	(*Rüstsatz 154 Rasterplattel*)
	ST03_418_B60_6: sDigInVisu;		(*  Zuführung links frei zum Ablegen ISK SP Maschine *)
	ST03_418_B60_7: sDigInVisu;		(*  Zuführung rechts frei zum Ablegen ISK SP Maschine *)

	ST03_419_B61_0: sDigInVisu;		(*  Förderband Zuführung links ISK anwesend zum Vereinzeln*)
	ST03_419_B61_1: sDigInVisu;		(*  Förderband Zuführung rechts ISK anwesend zum Vereinzeln*)
	ST03_419_B61_2: sDigInVisu;		(*  Züführung links ISK auf Übergabeposition Roboter Palettierer*)
	ST03_419_B61_3: sDigInVisu;		(*  Züführung rechts ISK auf Übergabeposition Roboter Palettierer*)

	ST03_419_Y61_5 : sValveVisu; 		(* Förderband linke Zuführung Vereinzler AST/GST *)
	ST03_419_Y61_6 : sValveVisu; 		(* Förderband rechte Zuführung Vereinzler AST/GST *)
	ST03_419_Y61_7 : sValveVisu; 		(* Förderband links/rechts Züführung Stopper AST/GST *)

	(*Rüstsatz 154pol*)

	ST03_425_B67_4: sDigInVisu;		(*  Zuführung  frei zum Ablegen ISK SP Maschine Pos.1 *)
	ST03_425_B67_5: sDigInVisu;		(*  Zuführung  frei zum Ablegen ISK SP Maschine Pos.2 *)
	ST03_425_B67_6: sDigInVisu;		(*  Zuführung  frei zum Ablegen ISK SP Maschine Pos.3 *)
	ST03_425_B67_7: sDigInVisu;		(*  ISK anwesend am Vereinzler*)

	ST03_426_B68_4: sDigInVisu;		(*  Züführung  ISK auf Übergabeposition Roboter Palettierer*)
	ST03_426_Y68_5 : sValveVisu; 		(* Förderband  Zuführung Vereinzler AST/GST *)
	ST03_426_Y68_6 : sValveVisu; 		(* Förderband  Züführung Stopper AST/GST *)


	(*Rüstsatz 160pol*)
	ST03_421_B63_4: sDigInVisu;		(*  Förderband frei zum Ablegen ISK SP Maschine Pos1 *)
	ST03_421_B63_5: sDigInVisu;		(*  Förderband frei zum Ablegen ISK SP Maschine Pos2 *)
	ST03_421_B63_6: sDigInVisu;		(*  Förderband frei zum Ablegen ISK SP Maschine Pos3 *)
	ST03_421_B63_7: sDigInVisu;		(*  ISK anwesend am Vereinzler*)
	ST03_422_B64_0: sDigInVisu;		(* Förderband Trigger Tintenstrahldrucker 1 (Lichtschranke)Rüstsatz*)
	ST03_423_B66_0: sDigInVisu;		(* Förderband Trigger Tintenstrahldrucker 2 (Lichtschranke) Rüstsatz*)
	ST03_8_B76_1: sDigInVisu;		(* Förderband Trigger Tintenstrahldrucker (Lichtschranke) 3621*)
	ST03_8_B76_2: sDigInVisu;		(* Förderband Trigger Tintenstrahldrucker (Lichtschranke) 3621*)
	ST03_422_B64_3: sDigInVisu;		(* Förderband ISK anwesend Stopper 1 Kamera*)
	ST03_423_B65_2: sDigInVisu;		(* Förderband ISK anwesend Stopper 2 Kamera*)
	ST03_423_B65_5: sDigInVisu;		(* Förderband ISK anwesend Stopper 3 Kamera*)
	ST03_422_B64_4: sDigInVisu; 		(* Zuführung ISK auf Übergabeposition Robo Palettierer*)

	ST03_422_Y64_5 : sValveVisu; 		(* Förderband  Zuführung Vereinzler AST/GST *)
	ST03_422_Y64_6 : sValveVisu; 		(* Förderband  Stopper Vereinzler AST/GST *)
	ST03_422_Y64_7 : sValveVisu; 		(* Förderband  Stopper 1 Kamera AST/GST *)
	ST03_423_Y65_6 : sValveVisu; 		(* Förderband  Stopper 2 Kamera AST/GST *)
	ST03_423_Y65_7 : sValveVisu; 		(* Förderband  Stopper 3 Kamera AST/GST *)

	ST03_33F4: sDigInVisu; 			(*Steckdosenleise Tintenstrahldrucker*)
	ST03_70U3_1: sDigInVisu; 			(*Bereit/ Im Druck Tintenstrahldrucker Frontseite*)
	ST03_70U3_2: sDigInVisu; 			(*Tank voll Tintenstrahldrucker Frontseite*)
	ST03_70U3_3: sDigInVisu; 			(*Fehler/Störung Tintenstrahldrucker Frontseite*)
	ST03_71U3_1: sDigInVisu; 			(*Bereit/ Im Druck Tintenstrahldrucker Rückseite*)
	ST03_71U3_2: sDigInVisu; 			(*Tank voll Tintenstrahldrucker Rückseite*)
	ST03_71U3_3: sDigInVisu; 			(*Fehler/Störung Tintenstrahldrucker Rückseite*)

	ST03_PLAN_70V1_1:sDigOutInVisu; 	(* Start  Bedrucken Tintenstrahldrucker Frontseite*)
	ST03_PLAN_71V1_2:sDigOutInVisu; 	(* Start  Bedrucken Tintenstrahldrucker Rückseite*)

	ST03_Y01 			: sValveVisu; 			(*1: Einschaltventil Hauptluft Tintenstrahldrucker nur bei SG-Maschine 3621*)
	ST03_S18			: sDigInVisu; 			(* ST02 Druckschalter Wartungseinheit Hauptluft min.6 bar *)
	ST03_H6 			: sDigOutInVisu; 		(* Signalsäule GR Bedruckung IO *)
	ST03_H7 			: sDigOutInVisu; 		(* Signalsäule RD Sammelstörung Bedruckung *)

	(*Rüstsatz 206pol*)

	ST03_435_B67_4: sDigInVisu;		(*  Zuführung  frei zum Ablegen ISK SP Maschine Pos.1 *)
(*	ST03_425_B67_5: sDigInVisu;		(*  Zuführung  frei zum Ablegen ISK SP Maschine Pos.2 *)
	ST03_425_B67_6: sDigInVisu;		(*  Zuführung  frei zum Ablegen ISK SP Maschine Pos.3 *) *)
	ST03_435_B67_7: sDigInVisu;		(*  ISK anwesend am Vereinzler*)

	ST03_436_B68_1: sDigInVisu;		(*  Züführung  ISK auf Übergabeposition Roboter Palettierer 1*)
	ST03_436_B68_2: sDigInVisu;		(*  Züführung  ISK auf Übergabeposition Roboter Palettierer 2*)
	ST03_437_B68_4: sDigInVisu;		(*  Züführung  ISK auf Übergabeposition Roboter Palettierer*)
	ST03_437_Y68_5 : sValveVisu; 		(* Förderband  Zuführung Vereinzler AST/GST *)
	ST03_437_Y68_6 : sValveVisu; 		(* Förderband  Züführung Stopper AST/GST *)

(*Rüstsatz92pol*)

	ST03_444_B69_4: sDigInVisu;		(*  Zuführung  frei zum Ablegen ISK SP Maschine Pos.1 *)
	ST03_444_B69_7: sDigInVisu;		(*  ISK anwesend am Vereinzler*)

	ST03_445_B70_1: sDigInVisu;		(*  Züführung  ISK auf Übergabeposition Roboter Palettierer 1*)
	ST03_445_B70_2: sDigInVisu;		(*  Züführung  ISK auf Übergabeposition Roboter Palettierer 2*)
	ST03_446_B70_4: sDigInVisu;		(*  Züführung  ISK auf Übergabeposition Roboter Palettierer*)
	ST03_446_Y70_5 : sValveVisu; 		(* Förderband  Zuführung Vereinzler AST/GST *)
	ST03_446_Y70_6 : sValveVisu; 		(* Förderband  Züführung Stopper AST/GST *)


(*Rüstsatz124pol*)

	ST03_451_B69_4: sDigInVisu;		(*  Zuführung  frei zum Ablegen ISK SP Maschine Pos.1 *)
	ST03_451_B69_7: sDigInVisu;		(*  ISK anwesend am Vereinzler*)

	ST03_452_B70_1: sDigInVisu;		(*  Züführung  ISK auf Übergabeposition Roboter Palettierer 1*)
	ST03_452_B70_2: sDigInVisu;		(*  Züführung  ISK auf Übergabeposition Roboter Palettierer 2*)
	ST03_453_B70_4: sDigInVisu;		(*  Züführung  ISK auf Übergabeposition Roboter Palettierer*)
	ST03_453_Y70_5 : sValveVisu; 		(* Förderband  Zuführung Vereinzler AST/GST *)
	ST03_453_Y70_6 : sValveVisu; 		(* Förderband  Züführung Stopper AST/GST *)

(*Rüstsatz46pol*)

	ST03_461_B69_4: sDigInVisu;		(*  Zuführung  frei zum Ablegen ISK SP Maschine Pos.1 *)
	ST03_461_B69_7: sDigInVisu;		(*  ISK anwesend am Stopper*)

	ST03_462_B70_0: sDigInVisu;		(*   Förderband  ISK anwesend Wender*)
	ST03_462_B70_1: sDigInVisu;		(*  Züführung  ISK auf Übergabeposition Roboter Palettierer Lageerkennung 1*)
	ST03_462_B70_2: sDigInVisu;		(*  Züführung  ISK auf Übergabeposition Roboter Palettierer Lageerkennung 2*)
	ST03_463_B70_7: sDigInVisu;		(*  Züführung  ISK auf Übergabeposition Roboter Palettierer *)

	ST03_464_Y71_0 : sValveVisu; 		(* Förderband  Zuführung Vereinzelner Wendestation AST/GST *)
	ST03_464_Y71_1 : sValveVisu; 		(* Förderband  Zuführung Zylinder Vakuumdüsen AST/GST *)
	ST03_464_Y71_2 : sValveVisu; 		(* Förderband  Zuführung Wendestation Einlauf / Auslauf *)
	ST03_464_Y71_3 : sValveVisu; 		(* Förderband  Zuführung Vereinzler AST/GST *)
	ST03_464_Y71_4 : sValveVisu; 		(* Förderband  Zuführung Stopper AST/GST *)
	ST03_464_Y71_5 : sValveVisu; 		(* Förderband  Zuführung Vakuumdüsen EIN/AUS *)
	ST03_464_B71_6: sDigInVisu;		(* Förderband  Vakuum vorhanden *)
 	ST03_464_B71_7: sDigInVisu;		(*Förderband  Staustrecke mitte voll *)

(*Rüstsatz NOX 5+6 pol*)

	ST03_4x2_B69_0: sDigInVisu;		(*Zuführung frei zum Ablegen ISK SP Maschine *)
	ST03_4x2_B69_5: sDigInVisu;		(* ISK anwesend am Stopper *)

	ST03_4x3_B70_0: sDigInVisu;		(* ISK anwesend Übergabeposition Stopper*)
	ST03_4x3_B70_1: sDigInVisu;		(* ISK anwesend Übergabeposition*)

	ST03_4x3_Y70_5 : sValveVisu; 	(* Zuführung Vereinzler AST/GST *)
	ST03_4x3_Y70_6 : sValveVisu; 	(* Zuführung Stopper AST/GST *)
	ST03_4x3_Y70_7 : sValveVisu; 	(* Zuführung Stopper Übergabeposition AST/GST *)

(*Rüstsatz NOX 4 pol*)
	ST03_491_B69_0: sDigInVisu;		(*  Zuführung  frei zum Ablegen ISK SP Maschine*)
	ST03_491_B69_5: sDigInVisu;		(*  ISK anwesend am Stoper*)
	ST03_491_B69_7: sDigInVisu;		(*  ISK auf Abholposition Robi*)

	ST03_492_Y70_0 : sValveVisu; 		(* Förderband  Zuführung Vereinzler AST/GST *)
	ST03_492_Y70_1 : sValveVisu; 		(* Förderband  Züführung Stopper AST/GST *)

(*Rüstsatz 88 pol*)
	ST03_501_B69_0: sDigInVisu;		(*  Zuführung  frei zum Ablegen ISK SP Maschine*)

	ST03_501_B69_5: sDigInVisu;		(*  ISK anwesend am Vereinzler*)
	ST03_501_B69_6: sDigInVisu;		(*  ISK anwesend am Stoper*)
	ST03_501_B69_7: sDigInVisu;		(*  ISK auf Abholposition Robi*)

	ST03_502_B70_0: sDigInVisu;		(*  ISK Lageerkennung*)
	ST03_502_Y70_1 : sValveVisu; 		(* Förderband  Zuführung Vereinzler AST/GST *)
	ST03_502_Y70_2 : sValveVisu; 		(* Förderband  Züführung Stopper AST/GST *)

(*Rüstsatz 7 pol*)
	ST03_512_XG1:    sDigInVisu;			(*  ISK in Rinne*)
	ST03_514_B71_7: sDigInVisu;		(*  Führungsschiene frei zum schwenken*)

	ST03_513_B70_4: sDigInVisu;		(*  ISK anwesend am Stoper*)
	ST03_513_B70_7: sDigInVisu;		(*  ISK auf Übergabeposition 1*)

	ST03_514_B71_2: sDigInVisu;		(*  ISK auf Übergabeposition 2*)
	ST03_514_B71_5: sDigInVisu;		(*  ISK auf Übergabeposition 3*)
	ST03_514_B71_6: sDigInVisu;		(*  ISK auf Übergabeposition 4*)

	ST03_515_Y72_0 : sValveVisu; 		(* SK Klemmen in Rinne AST/GST *)
	ST03_515_Y72_1 : sValveVisu; 		(* Rinne schwenkern AST/GST *)
	ST03_515_Y72_2 : sValveVisu; 		(* Führungsschiene  Zuführung Vereinzler AST/GST *)
	ST03_515_Y72_3 : sValveVisu; 		(* Führungsschiene  Zuführung Stopper AST/GST *)
	ST03_515_Y72_4 : sValveVisu; 		(* Übergabeposition Stopper 1  AST/GST *)
	ST03_515_Y72_5 : sValveVisu; 		(* Übergabeposition Stopper 2  AST/GST *)
	ST03_515_Y72_6 : sValveVisu; 		(* Übergabeposition Stopper 3  AST/GST *)

(*Rüstsatz 88 pol AMG*)
	ST03_521_B69_0: sDigInVisu;			(*Zuführung  frei zum Ablegen ISK SP Maschine*)

	ST03_521_B69_6: sDigInVisu;			(*ISK anwesend am Stopper*)
	ST03_521_B69_7: sDigInVisu;			(*ISK Lageerkennung links*)

	ST03_522_B70_0: sDigInVisu;			(*ISK Lageerkennung rechts*)
	ST03_522_Y70_1 : sValveVisu; 		(*Zuführung Vereinzler AST/GST *)
	ST03_522_Y70_2 : sValveVisu; 		(*Züführung Stopper AST/GST*)

(*Rüstsatz 120 pol *)
	ST03_531_B69_0: sDigInVisu;			(*Zuführung  frei zum Ablegen ISK SP Maschine*)

	ST03_531_B69_6: sDigInVisu;			(*ISK anwesend am Stopper*)
	ST03_531_B69_7: sDigInVisu;			(*ISK rechts Lageerkennung*)

	ST03_532_B70_0: sDigInVisu;			(*ISK links Lageerkennung *)
	ST03_532_Y70_1 : sValveVisu; 		(*Zuführung Vereinzler AST/GST *)
	ST03_532_Y70_2 : sValveVisu; 		(*Züführung Stopper AST/GST*)

(*Rüstsatz 21 pol *)
	ST03_536_B69_0: sDigInVisu;			(*Zuführung  frei zum Ablegen ISK SP Maschine*)

	ST03_536_B69_6: sDigInVisu;			(*ISK anwesend am Stopper*)
	ST03_536_B69_7: sDigInVisu;			(*ISK anwesend an Abholposition*)

	ST03_537_B70_0: sDigInVisu;			(*ISK Lageerkennung *)
	ST03_537_Y70_1 : sValveVisu; 		(*Zuführung Vereinzler AST/GST *)
	ST03_537_Y70_2 : sValveVisu; 		(*Züführung Stopper AST/GST*)

(*Rüstsatz 191 pol *)
	ST03_541_B69_0: sDigInVisu;			(*Zuführung  frei zum Ablegen ISK SP Maschine*)

	ST03_541_B69_6: sDigInVisu;			(*ISK anwesend am Stopper*)
	ST03_541_B69_7: sDigInVisu;			(*ISK rechts Lageerkennung*)

	ST03_542_B70_0: sDigInVisu;			(*ISK links Lageerkennung*)
	ST03_542_Y70_1 : sValveVisu; 		(*Zuführung Vereinzler AST/GST *)
	ST03_542_Y70_2 : sValveVisu; 		(*Züführung Stopper AST/GST*)

(*Rüstsatz  72pol *)
	ST03_546_B69_0: sDigInVisu;			(*Zuführung  frei zum Ablegen ISK SP Maschine*)

	ST03_546_B69_6: sDigInVisu;			(*ISK anwesend am Stopper*)
	ST03_546_B69_7: sDigInVisu;			(*ISK rechts Lageerkennung*)

	ST03_547_B70_0: sDigInVisu;			(*ISK links Lageerkennung*)
	ST03_547_Y70_1 : sValveVisu; 		(*Zuführung Vereinzler AST/GST *)
	ST03_547_Y70_2 : sValveVisu; 		(*Züführung Stopper AST/GST*)

(*Rüstsatz 48 pol *)
	ST03_551_B69_0: sDigInVisu;			(*Zuführung  frei zum Ablegen ISK SP Maschine*)

	ST03_551_B69_6: sDigInVisu;			(*ISK anwesend am Stopper*)
	ST03_551_B69_7: sDigInVisu;			(*ISK rechts Lageerkennung*)

	ST03_552_B70_0: sDigInVisu;		(*ISK links Lageerkennung*)
	ST03_552_Y70_1 : sValveVisu; 		(*Zuführung Vereinzler AST/GST *)
	ST03_552_Y70_2 : sValveVisu; 		(*Züführung Stopper AST/GST*)

(*Rüstsatz 268 pol *)
	ST03_556_B69_0: sDigInVisu;		(*Zuführung  frei zum Ablegen ISK SP Maschine*)

	ST03_556_B69_5: sDigInVisu;		(* Führungsschiene Überwachung Staustrecke*)
	ST03_556_B69_6: sDigInVisu;		(*ISK anwesend am Stopper*)
	ST03_556_B69_7: sDigInVisu;		(*ISK anwesend an Abholposition*)

	ST03_557_Y70_1 : sValveVisu; 		(*Zuführung Vereinzler AST/GST *)
	ST03_557_Y70_2 : sValveVisu; 		(*Züführung Stopper AST/GST*)

(*Rüstsatz 268 pol Rasterplatte======================================================================================*)
	ST03_562_B69_0: sDigInVisu;		(*Zuführung 1 frei zum schwenken*)
	ST03_562_B69_6: sDigInVisu;		(*Zuführung 1 ISK anwesend am Stopper*)
	ST03_562_B67_7: sDigInVisu;		(*Zuführung 1 ISK auf Übergabepos. Robi*)

	ST03_563_B70_0: sDigInVisu;		(*Zuführung 2 frei zum schwenken*)
	ST03_563_B70_6: sDigInVisu;		(*Zuführung 2 ISK anwesend am Stopper*)
	ST03_563_B70_7: sDigInVisu;		(*Zuführung 2 ISK auf Übergabepos. Robi*)

	ST03_564_Y71_0: sValveVisu; 		(*Zuführung 1 Vereinzler AST/GST *)
	ST03_564_Y71_1: sValveVisu; 		(*Zuführung 1 Stopper AST/GST *)
	ST03_564_Y71_2: sValveVisu; 		(*Zuführung 2 Vereinzler AST/GST *)
	ST03_564_Y71_3: sValveVisu; 		(*Zuführung 2 Stopper AST/GST *)
	ST03_564_Y71_4: sValveVisu; 		(* ISK Klemmer AST/GST *)
	ST03_564_Y71_5: sValveVisu; 		(* Rinne schwenkern AST/GST *)

	ST03_565_B72_0: sDigInVisu;		(* ISK 1 in Klemmer*)
	ST03_565_B72_1: sDigInVisu;		(* ISK 2 in Klemmer*)

(*Rüstsatz 33 pol Rasterplatte======================================================================================*)
	ST03_571_B69_0	: sDigInVisu;		(* Zuführung  Pos 1 frei zum Ablegen ISK SP Maschine*)
	ST03_571_B69_1	: sDigInVisu;		(* Zuführung  Pos 2 frei zum Ablegen ISK SP Maschine*)

	ST03_571_B69_6	: sDigInVisu;		(* ISK anwesend am Stopper*)
	ST03_571_B69_7	: sDigInVisu;		(* ISK anwesend an Abholposition*)

	ST03_572_Y70_0	: sValveVisu; 		(* Zuführung Vereinzler AST/GST *)
	ST03_572_Y70_1	: sValveVisu; 		(* Züführung Stopper AST/GST *)

(*---------------------------------------------------------------------------
  Station08
  ---------------------------------------------------------------------------*)


	ST08_170_Q2 : sDigInVisu; (* Bandstrecken Station 8 Motorschutz i.O. *)
	ST08_170_M : sDigInVisu; (* Bandstrecken Station 8 Thermokontakt i.O. *)

	ST08_400_B50_0 : sDigInVisu; (* Traystapel vor Vereinzeler Einlaufband hinten *)
	ST08_401_B50_5 : sDigInVisu; (* Traystapel vor Vereinzeler Einlaufband mitte *)
	ST08_402_B51_2 : sDigInVisu; (* Traystapel vor Vereinzeler Einlaufband vorne *)
	ST08_402_B51_4 : sDigInVisu; (* Luftzone 1 *)
	ST08_402_B51_5 : sDigInVisu; (* Luftzone 2 *)
	ST08_404_B52_2 : sDigInVisu; (* Traystapel in Ablageposition Isokörper *)
	ST08_404_B52_3 : sDigInVisu; (* Traystapel richtig eingelegt Isokörper *)
	ST08_406_B54_0 : sDigInVisu; (* Tray in Zwischenp. Entnahme Isokörper (Bandende) *)
	ST08_406_B54_3 : sDigInVisu; (* Tray in Ausheber. Entnahme Isokörper (Bandende) *)
	ST08_406_B54_6 : sDigInVisu; (* Tray aus Entnahme ausgelaufen (Bandende) *)
	ST08_407_B55_1 : sDigInVisu; (* Tray aus entnahme ausgelaufen STN8 *)
	ST08_407_B55_4 : sDigInVisu; (* Tray in Aufstapelposition eingelaufen STN8 *)
	ST08_409_B55_5 : sDigInVisu; (* Auslaufrollenbahn voll STN8 *)

	ST08_412_B58_4: sDigInVisu;		(*  Rüstsatz Förderband frei zum Ablegen ISK von SP Maschine Position 1 *)
	ST08_412_B58_5: sDigInVisu;		(*  Rüstsatz Förderband frei zum Ablegen ISK von SP Maschine Position 2 *)
	ST08_412_B58_6: sDigInVisu;		(*  Rüstsatz Förderband frei zum Ablegen ISK von SP Maschine Position 3 *)
	ST08_412_B58_5_35pol: sDigInVisu;		(*  Lageerkennung links *)
	ST08_412_B58_6_35pol: sDigInVisu;		(*  Lageerkennung rechts *)
	ST08_412_B58_7: sDigInVisu;		(*  Rüstsatz Förderband ISK anwesend zum Vereinzeln *)
	ST08_412_B59_0: sDigInVisu;		(*  Rüstsatz Förderband ISK auf Übergabeposition Roboter Verpackung *)

	ST08_169_K1 : sDigOutInVisu; (* Bandantrieb 1 Einlauf Trays Ein *)
	ST08_169_K2 : sDigOutInVisu; (* Bandantrieb 4 Auslauf leere Trays Ein *)
	ST08_170_K1 : sDigOutInVisu; (* Bandantrieb 2 Hubquereinheit Trays Ein *)
	ST08_170_K2 : sDigOutInVisu; (* Bandantrieb 3 Hubquereinheit Trays Ein *)

	ST08_400_Y50_0 : sValveVisu; (* Stopper Traystapel Einlaufb. hinten links + rechts AST *)
	ST08_400_Y50_2 : sValveVisu; (* Stopper Traystapel Einlaufb. mitte links + rechts AST *)
	ST08_402_Y50_4 : sValveVisu; (* Stopper Traystapel Einlaufb. vorne links + rechts AST *)
	ST08_403_Y50_6 : sValveVisu; (* Vakuum 1 Einlauf STN8 AST *)
	ST08_403_Y50_7 : sValveVisu; (* Vakuum 2 Einlauf STN8 AST *)
	ST08_405_Y51_0 : sValveVisu; (* Hubtüre 2 Einlauf Isokörper STN8 AST *)
	ST08_404_Y51_6 : sValveVisu; (* Stopper Traystapel Isokörper AST *)
	ST08_406_Y51_2 : sValveVisu; (* Hubtüre 3 STN8 AST *)
	ST08_407_Y51_4 : sValveVisu; (* Hubtüre 4 Auslauf STN8 AST *)
	ST08_404_Y52_0 : sValveVisu; (* Hub Bandstrecke AST *)
	ST08_406_Y52_3 : sValveVisu; (* Ausheber Trays Entnahmepos. Isok. STN8 GST *)
	ST08_401_Y52_4 : sValveVisu; (* Traystapel schieben hinte AST *)
	ST08_400_Y52_5 : sValveVisu; (* Stopper links + rechts Traystapel Auslaufband einfahren *)
	ST08_402_Y52_6 : sValveVisu; (* Traystapel schieben mitte AST *)
	ST08_402_Y52_7 : sValveVisu; (* Traystapel schieben vorne AST *)
	ST08_404_Y53_0 : sValveVisu; (* Abstapelzylinder 1 Isokörper AST *)
	ST08_404_Y53_2 : sValveVisu; (* Abstapelzylinder 2 Isokörper AST *)
	ST08_405_Y53_4 : sValveVisu; (* Rückhaltezylinder li+re Traystapel Isokörper AST *)
	ST08_408_Y54_0 : sValveVisu; (* Rückhaltezylinder li.+re. Auslauf STN8 AST *)
	ST08_408_Y54_2 : sValveVisu; (* Abstapelzylinder 1 STN8 AST *)
	ST08_408_Y54_4 : sValveVisu; (* Abstapelzylinder 2 STN8 AST *)

	ST08_412_Y55_0 : sValveVisu; (* Rüstsatz Förderband Vereinzelner *)
	ST08_412_Y55_2 : sValveVisu; (* Rüstsatz Förderband Stopper *)

	ST08_180_M1 		: sDigInVisu; (* Abstapeln *)
	ST08_185_M1 		: sDigInVisu; (* Aufstapeln *)
	ST08_190_M1 		: sDigInVisu; (* Tray ausheben *)

END_STRUCT
END_TYPE

(* Data type in System/LoginDialog *)
TYPE sVisuLoginDialog :
STRUCT

	LoginKeyPad			: sNumericKeypad;
	btn_Login			: sButtonVisu;
	btn_LogOut			: sButtonVisu;
	btn_ChangeUserData	: sButtonVisu;
	btn_ChangePassword	: sButtonVisu;

	ShowEditFields		: BOOL;
	UserListIndex		: INT;

	UserEdit			: sUserData;

END_STRUCT
END_TYPE

(* POU pBasic/PLC_PRG, ST *)
PROGRAM PLC_PRG
VAR_OUTPUT
	GlobalHomePos		: BOOL;
END_VAR
VAR
	DW_alive			: DINT:=0;
	TimeStart			: TIME;
	TimeEnd				: TIME;
	fb_ton_startHYDRA	: TON;
END_VAR
DW_alive:=DW_alive+1;
TimeStart:=TIME();

BusDiagnosis();
(*LngHandler();*)
IOSimulation();
ErrorHandler.ClearAll(sVisu:=Visu.ErrorHandler);
MessageHandler.ClearAll(sVisu:=Visu.Message);
IF	ProcessMessage01 = '' OR ProcessMessage02 = '' OR
	ModeSelect.Mode<=MODE_MANUAL THEN
	ProcessMessage01:='EMPTY';
	ProcessMessage02:='EMPTY';
END_IF

ModeSelect(	sVisu				:=Visu.ModeSelect,
			ControlOn			:= ST00_200_A1_A1.BitInToCheck,
 			SafetyDoorOk		:= gReadyForControlOn,
			MainValveOk			:= ST00_350_B20_0.BitInToCheck OR		SpecialMode03.State=STATE_RUN(* @@@ *),
			EmergencyOk			:= ST00_200_A1_A1.BitInToCheck,
			BusControlState		:= STATE_OK,
			UserOK				:= TRUE,
			AutoCycleEnd 		:= CheckSFCInInit.AllSeqInInit,
			SpecialCycleEnd 	:= CallSpecialModeSFCs.AllSpecialModeSFCInInit,
			HomePosRunEnd 		:= PLC_PRG.GlobalHomePos AND HomePositionSFC.State=STATE_WAIT,
			AllDoorsClosed 		:= TRUE,
			EnableFromPrevMach	:= TRUE,
			EnableFromNextMach	:= TRUE,
			ProtecKeyNotIn		:= TRUE,
			ProtecNotBridged	:= TRUE,
			Enable 			    := TRUE,
			Reset 				:= FALSE,
					);

gResetAll:=ModeSelect.QReset;

CallGeneralFunctions();
(* Spezialfunktion: *)
(* Disconnect Scanner TCPIP-Gateway *)
gBasicManualMode:=ModeSelect.BasicManualMode;

(*----------------------------------------------------------------------------
 Main-Program
 ----------------------------------------------------------------------------*)

ST_UPS(b_Ups := TRUE);
ST_CPU();
ST_AutoCheckIn( i_IntervalDay:=7 );
ST_MainMenue();
ST_Path();
ST_MinExit();
ST_ReadXmlLine();
ST_ReadXmlLineMsg();
ST_SaveAndLoad();
ST_Lng();

fb_ton_startHYDRA(IN:=TD.ArtNo <> '',PT:=t#5s);
IF fb_ton_startHYDRA.Q THEN						(*Textdateien erst nach Einlesen der Typdaten (Maschinennummer>0) + 5 sekündiger Verzögerung schreiben/lesen*)

	(***Für HYDRA 8****************************************)
	ST_Hydra8();

	FbExportHydraString(s_Path:= 'C:\MPDV\AIP2\spool\',
					st_data:=st_Hydra8Data,
					s_system_time:=gVarStrSystemTime,
					sDateiName:= 'Eingang.txt',
					bKopiereDateiAufServer:=FALSE,
					sToolPath := s_tools_path,
					tStartTime:= T#5S);

	ST_ImportHydraString(s_Path:= 'C:\MPDV\AIP2\spool\',
						sDateiName:= 'Ausgang.txt',
						tStartTime := T#5S);

END_IF

IF gInitOk AND ST_Path.Done THEN

	ImpExp_UD(path:= s_ud_path,filename:='UserData.xml');

	UserLoginHandler(sVisu:= Visu.LoginHandler,UserList:=UD.UserList);
	TDHandler(TDActivationAlowed:= ModeSelect.Mode<=MODE_MANUAL ,sVisu:=sTDHandler);
	MPHandler(sVisu:=sMPHandler);
	MP_ShiftHandler();

	ListHomeNOK(Clear:=TRUE);
	gHomeOk:=TRUE;
	_CallFBs();

	GlobalHomePos:=gHomeOk (*AND gHomePosSFCDone*);


	_CallSFCs();
	_CallPRGs();
	CheckSFCInInit();

ELSE
	gInitCollect:=TRUE;
	_CallInit();
	gInitOk:=gInitCollect;
 (* Spezialfunktion: *)
END_IF (*gInitOk=TRUE*)

(*------------- Main-Program-End -------------------------------------------*)

ErrorHandler.HandleErrors(sVisu:=Visu.ErrorHandler);
ErrorHandler.VisuUpdate(sVisu:=Visu.ErrorHandler);
MessageHandler.VisuUpdate(sVisu:=Visu.Message);

TimeEnd:=TIME();

(*END Program -----------------------------------------------------------------*)
END_PROGRAM

(* POU System/BusDiagnosis/BusDiagnosis, ST *)
PROGRAM BusDiagnosis
VAR

	EtheCatMasterAmsNetId 		AT %I* 	: ARRAY[0..5] OF USINT;	(* AmsNetId of EtherCat Mater *)


	GetConfSlaves				: FB_EcGetConfSlaves;			(* Read all Configured Informations of Master *)
	GetScannedSlaves			: FB_EcGetScannedSlaves;
	GetAllSlaveStates			: FB_EcGetAllSlaveStates;

	ConfSlaveInfo 				: ARRAY[1..NoOfMaxSlaves] OF ST_EcSlaveConfigData;
	ScannedSlaveInfo 			: ARRAY[1..NoOfMaxSlaves] OF ST_EcSlaveScannedData;
	ScannedSlaveInfoTemp 		: ARRAY[1..NoOfMaxSlaves] OF ST_EcSlaveScannedData;

	SlaveStates					: ARRAY[1..NoOfMaxSlaves] OF ST_EcSlaveState;
	SlaveStatesTemp			: ARRAY[1..NoOfMaxSlaves] OF ST_EcSlaveState;
	StringSlaveStates			: ARRAY[1..NoOfMaxSlaves] OF STRING(80);


	FirstStart					: BOOL;

	WorkIdx					: DINT;
	ForIdx						: DINT;

END_VAR
VAR CONSTANT
	NoOfMaxSlaves				: DINT := 100;
END_VAR
(* Get EtherCat Config - ONCE after RESET *)
IF 	NOT FirstStart THEN
	GetConfSlaves.bExecute:=TRUE;
	FirstStart:=TRUE;
END_IF

(* Get actual EtherCat - Scan *)
CASE WorkIdx OF
0: (* Init *)
	WorkIdx:=1;
1: (* Start Getting Bus Scan *)
	GetScannedSlaves.bExecute:=TRUE;
	IF 	GetScannedSlaves.bBusy THEN
		WorkIdx:=2;
	END_IF
2:
	IF 	NOT GetScannedSlaves.bBusy THEN
		WorkIdx:=3;
		ScannedSlaveInfo:=ScannedSlaveInfoTemp;
	END_IF

3:(* Get Salve States *)
	GetAllSlaveStates.bExecute:=TRUE;
	IF 	GetAllSlaveStates.bBusy THEN
		WorkIdx:=4;
	END_IF
4:
	IF 	NOT GetAllSlaveStates.bBusy THEN
		WorkIdx:=5;
		SlaveStates:=SlaveStatesTemp;
		FOR ForIdx:=1 TO NoOfMaxSlaves DO
			StringSlaveStates[ForIdx]:=F_ConvSlaveStateToString(SlaveStates[ForIdx]);
		END_FOR
	END_IF
5: (* End of operation *)
	WorkIdx:=0;
END_CASE

GetConfSlaves(
	sNetId					:= GetAmsNetIdString(EtheCatMasterAmsNetId),
	pArrEcConfSlaveInfo		:= ADR(ConfSlaveInfo),
	cbBufLen				:= SIZEOF(ConfSlaveInfo),
);

GetConfSlaves.bExecute:=FALSE;

GetScannedSlaves(
	sNetId						:= GetAmsNetIdString(EtheCatMasterAmsNetId),
	pArrEcScannedSlaveInfo	:= ADR(ScannedSlaveInfoTemp),
	cbBufLen					:= SIZEOF(ScannedSlaveInfoTemp),
 );

GetScannedSlaves.bExecute:=FALSE;

GetAllSlaveStates(
	sNetId						:= GetAmsNetIdString(EtheCatMasterAmsNetId),
	pStateBuf					:= ADR(SlaveStatesTemp),
	cbBufLen					:= ADR(SlaveStatesTemp),
 );

GetAllSlaveStates.bExecute:=FALSE;
END_PROGRAM

(* POU System/BusDiagnosis/GetAmsNetIdString, ST *)
FUNCTION GetAmsNetIdString : STRING
VAR_INPUT
		EtheCatMasterAmsNetId : ARRAY[0..5] OF USINT;
END_VAR
VAR
	Idx : DINT;
END_VAR
GetAmsNetIdString:='';

FOR Idx:=0 TO 5 DO
	GetAmsNetIdString:=CONCAT(GetAmsNetIdString, USINT_TO_STRING(EtheCatMasterAmsNetId[Idx]));
	IF 	Idx<>5 THEN
		GetAmsNetIdString:=CONCAT(GetAmsNetIdString,'.');
	END_IF
END_FOR
END_FUNCTION

(* POU Stations/ST_00/ST00_PRGs/IOSimulation, ST *)
PROGRAM IOSimulation
VAR

END_VAR
SystemTaskInfoArr[1].cycleTimeExceeded;
SystemTaskInfoArr[1].lastExecTime;
END_PROGRAM

(* POU System/Error_and_Message/ErrorHandler, ST *)
PROGRAM ErrorHandler
VAR
	TempErrorArray					: sErrorHandlerVisu;
	TempErrorArrayLastCycle 		: sErrorHandlerVisu;
	TempErrorArrayLastCycleQuitt 	: sErrorHandlerVisu;
	Idx								: DINT;

	TempError						: BOOL;
	TempWarning					: BOOL;
	TempInfo						: BOOL;
	POS							: INT;
	i								: INT;

	(* Variable for ErrorHistory Handling *)
	Idx_Akt							: DINT;
	Idx_Last						: DINT;
	ErrorPresent						:BOOL;

	CompareValue					:DINT;

	(* Variables for ErrorLog.CSV *)
	ErrorLogBuffer				: ARRAY[0..100] OF ErrorStruct;
	EmptyError					: ErrorStruct;
	ErrorToLog					: ErrorStruct;
	ErrorToQuitt					: ErrorStruct;

	StepExportError				: DINT;

	(* CSV Config *)
	ColIdx						: DINT;
	DataType					: DataTypeDef;
	CSVConfig  					: ARRAY[1..20] OF CSV_Config;
	CSVConfigDone				: BOOL :=FALSE;
	ErrorExport					: CSVExport_AppendLineWithVarConfig;				(*Daten in CSV-Datei exportieren*)
END_VAR
VAR_INPUT
	ErrorLogFileName			: STRING(255) := ''; (* Filename with Path e.g. 'C:\ErrorLog.csv' *)
	ErrorToAdd					: ErrorStruct;
END_VAR
VAR_OUTPUT
	bOutError					: BOOL;
	bOutWarning				: BOOL;
	bOutInfo					: BOOL;
END_VAR
VAR_IN_OUT
	sVisu						: sErrorHandlerVisu;
END_VAR
;
END_PROGRAM
ACTION AddError:
FOR Idx:=0 TO NO_OF_ERRORS
DO

	IF TempErrorArray.Error[Idx].No=0
	THEN

		FOR i:=0 TO 5 DO	(*Leerstellen entfernen*)
			POS:=0;
			POS := FIND (ErrorToAdd.Text,'$R');
			IF POS <> 0 THEN
				ErrorToAdd.Text := DELETE (ErrorToAdd.Text,1,POS);
			END_IF
			POS:=0;
			POS := FIND (ErrorToAdd.Text,'$N');
			IF POS <> 0 THEN
				ErrorToAdd.Text := DELETE (ErrorToAdd.Text,1,POS);
			END_IF
		END_FOR

		TempErrorArray.Error[Idx]:=ErrorToAdd;
			CASE TempErrorArray.Error[Idx].Typ OF
				0: TempErrorArray.Error[Idx].LineColor:=color.salmon;
				1: TempErrorArray.Error[Idx].LineColor:=color.orange;
				2: TempErrorArray.Error[Idx].LineColor:=color.lightblue;
			END_CASE
		EXIT;
	END_IF
END_FOR
END_ACTION
ACTION ClearAll:
FOR Idx:=0 TO NO_OF_ERRORS
DO
	TempErrorArray.Error[Idx].No:=0;
	TempErrorArray.Error[Idx].No:=0;
	TempErrorArray.Error[Idx].DateTime:=DINT_TO_DT(0);
	TempErrorArray.Error[Idx].Text:='';
	TempErrorArray.Error[Idx].Typ:=0;
	TempErrorArray.Error[Idx].Station:=0;
	TempErrorArray.Error[Idx].Prio:=0;
	TempErrorArray.Error[Idx].QuitAddr:=0;
END_FOR
END_ACTION
ACTION HandleErrors:
TempError			:= FALSE;
TempWarning		:= FALSE;
TempInfo			:= FALSE;

FOR Idx:=0 TO NO_OF_ERRORS
DO
	IF TempErrorArray.Error[Idx].No<>0 AND TempErrorArray.Error[Idx].Typ=0 AND NOT TempError
	THEN
		TempError:=TRUE;
	END_IF
	IF TempErrorArray.Error[Idx].No<>0 AND TempErrorArray.Error[Idx].Typ=1 AND NOT TempWarning
	THEN
		TempWarning:=TRUE;
	END_IF
	IF TempErrorArray.Error[Idx].No<>0 AND TempErrorArray.Error[Idx].Typ=2 AND NOT TempInfo
	THEN
		TempInfo:=TRUE;
	END_IF
END_FOR

bOutError:=TempError;
bOutWarning:=TempWarning;
bOutInfo:=TempInfo;

(*Eintrag in die Errorlog, wenn der Fehler wieder weggeht-----------------------------------------------------------------------------------------------------------------*)
IF MEMCMP(ADR(TempErrorArray.Error), ADR(TempErrorArrayLastCycleQuitt.Error), SIZEOF(TempErrorArray.Error))<>0 THEN
	ErrorToQuitt:=EmptyError;
	FOR Idx_Akt:=0 TO NO_OF_ERRORS DO

		FOR Idx_Last:=0 TO NO_OF_ERRORS DO
			IF	(*TempErrorArrayLastCycleQuitt.Error[Idx_Akt].DateTime = TempErrorArray.Error[Idx_Last].DateTime AND*)
				TempErrorArrayLastCycleQuitt.Error[Idx_Akt].Text = TempErrorArray.Error[Idx_Last].Text OR
				(*Ausnahmen*)
				FIND(TempErrorArrayLastCycleQuitt.Error[Idx_Akt].Text, 'MessageHandler') >0 OR
				FIND(TempErrorArrayLastCycleQuitt.Error[Idx_Akt].Text, 'TD') >0 OR
				FIND(TempErrorArrayLastCycleQuitt.Error[Idx_Akt].Text, 'Mode') >0 OR
				FIND(TempErrorArrayLastCycleQuitt.Error[Idx_Akt].Text, 'LoginHandler') >0 THEN
				EXIT;
			END_IF
		END_FOR

		IF 	Idx_Last >NO_OF_ERRORS THEN
			ErrorToQuitt:=TempErrorArrayLastCycleQuitt.Error[Idx_Akt];
			ErrorToQuitt.DateTime:=gVarDTSystemtime;
			ErrorToQuitt.Text:=CONCAT('quitt ',ErrorToQuitt.Text);

			IF ErrorLogFileName<>'' THEN
				FOR Idx:= 100 TO 2 BY -1 DO
					ErrorLogBuffer[Idx]:=ErrorLogBuffer[Idx-1];
				END_FOR
				ErrorLogBuffer[1]:=ErrorToQuitt;
			END_IF
		END_IF

	END_FOR
END_IF
TempErrorArrayLastCycleQuitt:= TempErrorArray;
(*-------------------------------------------------------------------------------------------------------------------------------------------------------------------------------------------------------*)

(* Handle Error History *)

IF MEMCMP(ADR(TempErrorArray.Error), ADR(TempErrorArrayLastCycle.Error), SIZEOF(TempErrorArray.Error))<>0
THEN
	FOR Idx_Akt:=0 TO NO_OF_ERRORS
	DO
		ErrorPresent:=FALSE;
		FOR Idx_Last:=0 TO NO_OF_ERRORS
		DO
			CompareValue:=MEMCMP(ADR(TempErrorArray.Error[Idx_Akt].DateTime), ADR(TempErrorArrayLastCycle.Error[Idx_Last].DateTime), SIZEOF(TempErrorArray.Error[Idx_Akt].DateTime));
			IF TempErrorArray.Error[Idx_Akt].DateTime = TempErrorArrayLastCycle.Error[Idx_Last].DateTime
			THEN
				ErrorPresent:=TRUE;
				EXIT;
			END_IF
		END_FOR
		(* Error is not present in List *)
		IF NOT ErrorPresent AND TempErrorArray.Error[Idx_Akt].No<>0
		THEN
			(* Add To ErrorHistory *)
			FOR Idx:= 500 TO 2 BY -1
			DO
				ErrorHistory[Idx]:=ErrorHistory[Idx-1];
			END_FOR
			ErrorHistory[1]:=TempErrorArray.Error[Idx_Akt];
			(* Add To Error Log Buffer *)
			IF ErrorLogFileName<>''
				THEN
				FOR Idx:= 100 TO 2 BY -1
				DO
					ErrorLogBuffer[Idx]:=ErrorLogBuffer[Idx-1];
				END_FOR
				ErrorLogBuffer[1]:=TempErrorArray.Error[Idx_Akt];
			END_IF

		END_IF
	END_FOR
END_IF

TempErrorArrayLastCycle:= TempErrorArray;


IF visu.ErrorHistoryScroll>470 THEN
visu.ErrorHistoryScroll:=0;
END_IF

IF visu.ErrorHistoryScroll<0 THEN
visu.ErrorHistoryScroll:=0;
END_IF

FOR Idx:=0 TO NO_OF_ERRORS
DO
	IF	(Idx+visu.ErrorHistoryScroll) <= NO_OF_ERRORS THEN
		Visu.ErrorHistory.Error[Idx]:=ErrorHistory[Idx+visu.ErrorHistoryScroll];
		Visu.ErrorHistory.Error[Idx].No:=Idx+visu.ErrorHistoryScroll;
	END_IF
END_FOR

ErrorHandler.WriteErrorLog;
END_ACTION
ACTION VisuUpdate:
sVisu.Error:=TempErrorArray.Error;

(*
Das muss noch folgendermaßen umgesetzt werden.
(g.baiz, am 03.03.2010)

Das Visu-Array wird dem TempErrorArray abgeglichen,
d.h. für jeden Fehler wird "ObjektName" und "Fehlernummer" verglichen.

- Wenn Fehler noch in Visu aber nicht mehr in TempErrorArray, dann in Visu löschen
- Wenn Fehler bereits in Visu und noch im TempErrorArray, dann nur den "ErrorText" nochmals in die Visu kopieren 
  (könnte sich bei gleicher Fehlernummer geändert haben)
- Wenn Fehler noch nicht in Visu aber in TempErrorArray, dann Zeitstempel eintragen und in Visu kopieren

*)
END_ACTION
ACTION WriteErrorLog:
(* Config Log File *)
IF NOT CSVConfigDone
THEN
	ColIdx:=1;
	CSVConfig[ColIdx].ColName				:=	'Nr';
	CSVConfig[ColIdx].ColDataType		:=	DataType.iDINT;
	CSVConfig[ColIdx].ColSourceAdr		:=	ADR(ErrorToLog.No);
	CSVConfig[ColIdx].ColSourceSize	:=	SIZEOF(ErrorToLog.No);

	ColIdx:=ColIdx+1;
	CSVConfig[ColIdx].ColName				:=	'Datum/Uhrzeit';
	CSVConfig[ColIdx].ColDataType		:=	DataType.iDT;
	CSVConfig[ColIdx].ColSourceAdr		:=	ADR(ErrorToLog.DateTime);
	CSVConfig[ColIdx].ColSourceSize	:=	SIZEOF(ErrorToLog.DateTime);
	
	ColIdx:=ColIdx+1;
	CSVConfig[ColIdx].ColName				:=	'Beschreibung';
	CSVConfig[ColIdx].ColDataType		:=	DataType.iSTRING;
	CSVConfig[ColIdx].ColSourceAdr		:=	ADR(ErrorToLog.Text);
	CSVConfig[ColIdx].ColSourceSize	:=	SIZEOF(ErrorToLog.Text);
	
	ColIdx:=ColIdx+1;
	CSVConfig[ColIdx].ColName				:=	'Typ';
	CSVConfig[ColIdx].ColDataType		:=	DataType.iDINT;
	CSVConfig[ColIdx].ColSourceAdr		:=	ADR(ErrorToLog.Typ);
	CSVConfig[ColIdx].ColSourceSize	:=	SIZEOF(ErrorToLog.Typ);
	
	CSVConfigDone:=TRUE;
END_IF

(* Add To Error Log File *)
IF ErrorLogFileName<>''
THEN

	(* Check Error to Log present when Export inactive *)
	IF StepExportError = 0 THEN

		FOR Idx:= 1 TO 100
		DO
			IF ErrorLogBuffer[Idx].DateTime=EmptyError.DateTime
			THEN
				IF Idx>1
				THEN
					ErrorToLog:=ErrorLogBuffer[Idx-1];
					ErrorLogBuffer[Idx-1]:=EmptyError;
					StepExportError:=1;
				END_IF
				EXIT;
			END_IF
		END_FOR

	END_IF

	(* Export Error to specified CSV-File *)
	CASE StepExportError OF
	1: 	ErrorExport.nInExport:=TRUE;
		 	StepExportError:=2;
	2: 	IF ErrorExport.Done
			THEN
				StepExportError:=0;
			END_IF
	END_CASE

(* CylicCall *)
			ErrorExport(CSVConfig:=CSVConfig ,
									OverwriteExistingFile:=FALSE,
									strInFileName:=ErrorLogFileName ,
									localAMSNetID:= '',
									iInNumberOfColumns:= 4,
									CreateHeaderLine:=TRUE
									);

IF ErrorExport.Done
THEN
	ErrorExport.nInExport:=FALSE;
END_IF


END_IF
END_ACTION

(* POU zLibrary/CSV_ImportExport/CSVExport_AppendLineWithVarConfig, ST *)
FUNCTION_BLOCK CSVExport_AppendLineWithVarConfig
VAR_INPUT
	CSVConfig			: ARRAY[1..20] OF CSV_Config;
	nInExport			: BOOL;
	OverwriteExistingFile	: BOOL;
	strInFileName		: STRING(255);
	localAMSNetID		: T_AmsNetId;
	iInNumberOfColumns	: DINT;
	CreateHeaderLine	: BOOL;
END_VAR
VAR_OUTPUT
	Done				: BOOL;
END_VAR
VAR
	WorkingStep			: INT;
	WorkingStepWriteLine: INT;

	FindFile_			: FB_EnumFindFileEntry;
	filesList_			: ST_FindFileEntry;

	ActCol				: DINT;
	ActVarConfig		: CSV_Config;
	ActVarValueString	: STRING;
	AdressOffset		: DINT;

	FPStart				: R_TRIG;
	FNStart				: F_TRIG;

	FBFileOpen			: FB_FileOpen;
	nOpenMode			: DWORD;
	hHandle				: UINT;

	CreateHeaderLineNow:BOOL;

	FBFileWrite			: FB_FileWrite;
	FBFileClose			: FB_FileClose;
	FileOpenWasBusy		: BOOL;
	FileWriteWasBusy	: BOOL;
	FileCloseWasBusy	: BOOL;
	FileOpenStart		: BOOL;
	FileWriteStart		: BOOL;
	FileCloseStart		: BOOL;

	TempString			: STRING[255];
END_VAR
FPStart(CLK:= nInExport );
FNStart(CLK:= nInExport );

IF 	FPStart.Q THEN
	WorkingStep:=1;
	FileOpenWasBusy:=FALSE;
	FileWriteWasBusy:=FALSE;
	FileCloseWasBusy:=FALSE;
	FileOpenStart:=FALSE;
	FileWriteStart:=FALSE;
	FileCloseStart:=FALSE;
	WorkingStepWriteLine:=1;
	TempString:='';
END_IF;

IF 	FNStart.Q AND WorkingStep<>50 THEN
	WorkingStep:=0;
END_IF


CASE WorkingStep OF

	1:	(* Check File Exist *)
		FindFile_.bExecute:=TRUE;
		IF 	FindFile_.bBusy THEN
			WorkingStep:=2;
		END_IF
	2:
		FindFile_.bExecute:=TRUE;
		IF 	NOT FindFile_.bBusy THEN
			WorkingStep:=3;
		END_IF
	3:
		IF  	filesList_.sFileName='' THEN
			(* Create Header *)
			WorkingStep:=20;
			CreateHeaderLineNow:=CreateHeaderLine;
		ELSIF
			filesList_.sFileName<>'' THEN
			(* File Exists *)
			WorkingStep:=20;
			CreateHeaderLineNow:=FALSE;
		END_IF

	20: (* Open File *)
		IF 	OverwriteExistingFile THEN
			nOpenMode:=FOPEN_MODEWRITE OR FOPEN_MODETEXT ;
		ELSE
			nOpenMode:=FOPEN_MODEAPPEND OR FOPEN_MODETEXT ;
		END_IF
		FBFileOpen(
			sNetId			:= localAMSNetID,
			sPathName	:= strInFileName,
			nMode			:= nOpenMode,
			ePath			:= PATH_GENERIC,
			bExecute		:= FileOpenStart,
			tTimeout		:= t#1s);
			hHandle:=FBFileOpen.hFile;
		FileOpenStart:= TRUE;
		IF 	FBFileOpen.bBusy THEN
			FileOpenWasBusy:=TRUE;
		END_IF
		IF 	NOT FBFileOpen.bBusy AND FileOpenWasBusy THEN
			WorkingStep:=21;
			FileOpenStart:= FALSE;
		END_IF

	21:	(* Write Header if required *)
		IF 	CreateHeaderLineNow THEN
			IF 	WorkingStepWriteLine=0 THEN
				WorkingStepWriteLine:=0;
				TempString:='';
			END_IF

			CASE WorkingStepWriteLine OF
				0: (*Create new CSV config*)
						WorkingStepWriteLine:=1;
				1: (* Open File *)
					FOR ActCol := 1 TO iInNumberOfColumns DO
						(*CSV-Configuration zuweisen*)
						ActVarConfig:=CSVConfig[ActCol];
						TempString:=CONCAT(TempString,ActVarConfig.ColName);
						IF 	ActCol<iInNumberOfColumns THEN
							TempString:=CONCAT(TempString,';');
						ELSE
							TempString:=CONCAT(TempString, '$N');
						END_IF
					END_FOR;
					WorkingStepWriteLine:=2;
				2:(* Write Line *)
				FBFileWrite(
					sNetId				:=localAMSNetID ,
					hFile				:=hHandle ,
					pWriteBuff			:=ADR(TempString) ,
					cbWriteLen			:=LEN(TempString) ,
					bExecute			:=FileWriteStart ,
					tTimeout				:=t#1s );
					FileWriteStart			:= TRUE;
	
				IF 	FBFileWrite.bBusy  THEN
					FileWriteWasBusy:=TRUE;
				END_IF
				IF 	(NOT FBFileWrite.bBusy) AND FileWriteWasBusy THEN
					FileWriteStart:= FALSE;
					FileWriteWasBusy:=FALSE;

					WorkingStepWriteLine:=0;
					WorkingStep:=30;
				END_IF
			END_CASE
		ELSE
			WorkingStep:=30;
		END_IF

	30:	(* Write Data *)
		IF 	WorkingStepWriteLine=0 THEN
			WorkingStepWriteLine:=0;
			TempString:='';
		END_IF

		CASE WorkingStepWriteLine OF
			0: (*Create new CSV config*)
					WorkingStepWriteLine:=1;
			1: (* Open File *)
				FOR ActCol := 1 TO iInNumberOfColumns DO
					(*CSV-Configuration zuweisen*)
					ActVarConfig:=CSVConfig[ActCol];
					AdressOffset:=0;
					ActVarValueString:=TYPEDEF_TO_STRING(ActVarConfig,AdressOffset);
					TempString:=CONCAT(TempString,ActVarValueString);
					IF 	ActCol<iInNumberOfColumns THEN
						TempString:=CONCAT(TempString,';');
					ELSE
						TempString:=CONCAT(TempString, '$N');
					END_IF
				END_FOR
				WorkingStepWriteLine:=2;
			2:(* Write Line *)
			FBFileWrite(
				sNetId				:=localAMSNetID ,
				hFile				:=hHandle ,
				pWriteBuff			:=ADR(TempString) ,
				cbWriteLen			:=LEN(TempString) ,
				bExecute			:=FileWriteStart ,
				tTimeout				:=t#1s );
				FileWriteStart			:= TRUE;

			IF 	FBFileWrite.bBusy  THEN
				FileWriteWasBusy:=TRUE;
			END_IF
			IF 	(NOT FBFileWrite.bBusy) AND FileWriteWasBusy THEN
				FileWriteStart:= FALSE;
				FileWriteWasBusy:=FALSE;

				WorkingStepWriteLine:=0;
				WorkingStep:=40;

			END_IF
		END_CASE

	40: (* Close File *)
		FBFileClose(
			sNetId:=localAMSNetID ,
			hFile:= hHandle,
			bExecute:=FileCloseStart ,
			tTimeout:= t#1s);
		FileCloseStart:=TRUE;
		IF 	FBFileClose.bBusy THEN
			FileCloseWasBusy:=TRUE;
		END_IF

		IF 	NOT FBFileClose.bBusy AND FileCloseWasBusy THEN
			WorkingStep:=50;
		END_IF
	50:(* Done *)
		Done:=TRUE;
		IF 	FNStart.Q THEN
			WorkingStep:=0;
			done:=FALSE;
		END_IF

END_CASE

FindFile_(
	sNetId:= '',
	sPathName:= strInFileName,
	stFindFile=> filesList_
);

FindFile_.bExecute:=FALSE;
END_FUNCTION_BLOCK

(* POU zLibrary/CSV_ImportExport/TYPEDEF_TO_STRING, ST *)
FUNCTION TYPEDEF_TO_STRING : STRING
VAR_INPUT
	TypeData				:CSV_Config;
	inAdressOffset			:DINT;
END_VAR
VAR
	pBOOL					:POINTER TO 	BOOL;
	pBYTE					:POINTER TO 	BYTE;
	pWORD				:POINTER TO 	WORD;
	pDWORD				:POINTER TO 	DWORD;
	pSINT					:POINTER TO 	SINT;
	pUSINT					:POINTER TO USINT;
	pINT					:POINTER TO INT;
	pUINT					:POINTER TO UINT;
	pDINT					:POINTER TO DINT;
	pUDINT				:POINTER TO UDINT;
	pREAL					:POINTER TO REAL;
	pLREAL				:POINTER TO LREAL;
	pSTRING				:POINTER TO STRING(255);
	pTIME					:POINTER TO TIME;
	pTOD					:POINTER TO TOD;
	pDATE					:POINTER TO DATE;
	pDT					:POINTER TO DT;
END_VAR
VAR CONSTANT
	TempTypeData			:DataTypeDef;
END_VAR
IF 	TypeData.ColDataType = TempTypeData.iBOOL THEN
	pBOOL:=TypeData.ColSourceAdr + inAdressOffset;
	TYPEDEF_TO_STRING:=BOOL_TO_STRING(pBOOL^);
ELSIF
	TypeData.ColDataType = TempTypeData.iBYTE THEN
	pBYTE:=TypeData.ColSourceAdr + inAdressOffset;
	TYPEDEF_TO_STRING:=BYTE_TO_STRING(pBYTE^);
ELSIF
	TypeData.ColDataType = TempTypeData.iWORD THEN
	pWORD:=TypeData.ColSourceAdr + inAdressOffset;
	TYPEDEF_TO_STRING:=WORD_TO_STRING(pWORD^);
ELSIF
	TypeData.ColDataType = TempTypeData.iDWORD THEN
	pDWORD:=TypeData.ColSourceAdr + inAdressOffset;
	TYPEDEF_TO_STRING:=DWORD_TO_STRING(pDWORD^);
ELSIF
	TypeData.ColDataType = TempTypeData.iSINT THEN
	pSINT:=TypeData.ColSourceAdr + inAdressOffset;
	TYPEDEF_TO_STRING:=SINT_TO_STRING(pSINT^);
ELSIF
	TypeData.ColDataType = TempTypeData.iUSINT THEN
	pUSINT:=TypeData.ColSourceAdr + inAdressOffset;
	TYPEDEF_TO_STRING:=USINT_TO_STRING(pUSINT^);
ELSIF
	TypeData.ColDataType = TempTypeData.iINT THEN
	pINT:=TypeData.ColSourceAdr + inAdressOffset;
	TYPEDEF_TO_STRING:=INT_TO_STRING(pINT^);
ELSIF
	TypeData.ColDataType = TempTypeData.iUINT THEN
	pUINT:=TypeData.ColSourceAdr + inAdressOffset;
	TYPEDEF_TO_STRING:=UINT_TO_STRING(pUINT^);
ELSIF
	TypeData.ColDataType = TempTypeData.iDINT THEN
	pDINT:=TypeData.ColSourceAdr + inAdressOffset;
	TYPEDEF_TO_STRING:=DINT_TO_STRING(pDINT^);
ELSIF
	TypeData.ColDataType = TempTypeData.iUDINT THEN
	pUDINT:=TypeData.ColSourceAdr + inAdressOffset;
	TYPEDEF_TO_STRING:=UDINT_TO_STRING(pUDINT^);
ELSIF
	TypeData.ColDataType = TempTypeData.iREAL THEN
	pREAL:=TypeData.ColSourceAdr + inAdressOffset;
	TYPEDEF_TO_STRING:=REAL_TO_STRING(pREAL^);
ELSIF
	TypeData.ColDataType = TempTypeData.iLREAL THEN
	pLREAL:=TypeData.ColSourceAdr + inAdressOffset;
	TYPEDEF_TO_STRING:=LREAL_TO_STRING(pLREAL^);
ELSIF
	TypeData.ColDataType = TempTypeData.iSTRING THEN
	pSTRING:=TypeData.ColSourceAdr + inAdressOffset;
	IF 	pSTRING^='' THEN
		TYPEDEF_TO_STRING:='empty';
	ELSE
		TYPEDEF_TO_STRING:=pSTRING^;
	END_IF
ELSIF
	TypeData.ColDataType = TempTypeData.iTIME THEN
	pTIME:=TypeData.ColSourceAdr + inAdressOffset;
	TYPEDEF_TO_STRING:=TIME_TO_STRING(pTIME^);
ELSIF
	TypeData.ColDataType = TempTypeData.iTOD THEN
	pTOD:=TypeData.ColSourceAdr + inAdressOffset;
	TYPEDEF_TO_STRING:=TOD_TO_STRING(pTOD^);
ELSIF
	TypeData.ColDataType = TempTypeData.iDATE THEN
	pDATE:=TypeData.ColSourceAdr + inAdressOffset;
	TYPEDEF_TO_STRING:=DATE_TO_STRING(pDATE^);
ELSIF
	TypeData.ColDataType = TempTypeData.iDT THEN
	pDT:=TypeData.ColSourceAdr + inAdressOffset;
	TYPEDEF_TO_STRING:=DT_TO_SPECIALSTRING(pDT^);
ELSE
	TYPEDEF_TO_STRING:='error';
END_IF
END_FUNCTION

(* POU zLibrary/CSV_ImportExport/DT_TO_SPECIALSTRING, ST *)
FUNCTION DT_TO_SPECIALSTRING : STRING
VAR_INPUT
	inDT			:DT;
END_VAR
VAR
	TempString		:STRING;
	SysTime		:TIMESTRUCT;

	wYear			:WORD;
	wMonth			:WORD;
	wDay			:WORD;
	wHour			:WORD;
	wMin			:WORD;
	wSec			:WORD;
END_VAR
SysTime:=DT_TO_SYSTEMTIME(inDT);
wYear:=SysTime.wYear;
wMonth:=SysTime.wMonth;
wDay:=SysTime.wDay;
wHour:=SysTime.wHour;
wMin:=SysTime.wMinute;
wSec:=SysTime.wSecond;
TempString:='';

IF 	wDay<10 THEN
	TempString:=CONCAT(TempString ,WORD_TO_STRING(0));
END_IF
TempString:=CONCAT(TempString ,WORD_TO_STRING(wDay));
TempString:=CONCAT(TempString , '.');
IF 	wMonth<10 THEN
	TempString:=CONCAT(TempString ,WORD_TO_STRING(0));
END_IF
TempString:=CONCAT(TempString ,WORD_TO_STRING(wMonth));
TempString:=CONCAT(TempString , '.');
TempString:=CONCAT(TempString ,WORD_TO_STRING(wYear));
TempString:=CONCAT(TempString , ' ');
IF 	wHour<10 THEN
	TempString:=CONCAT(TempString ,WORD_TO_STRING(0));
END_IF
TempString:=CONCAT(TempString ,WORD_TO_STRING(wHour));
TempString:=CONCAT(TempString , ':');
IF 	wMin<10 THEN
	TempString:=CONCAT(TempString ,WORD_TO_STRING(0));
END_IF
TempString:=CONCAT(TempString ,WORD_TO_STRING(wMin));
TempString:=CONCAT(TempString , ':');
IF	wSec<10 THEN
	TempString:=CONCAT(TempString ,WORD_TO_STRING(0));
END_IF
TempString:=CONCAT(TempString ,WORD_TO_STRING(wSec));
DT_TO_SPECIALSTRING:=TempString;
END_FUNCTION

(* POU System/Error_and_Message/MessageHandler, ST *)
PROGRAM MessageHandler
VAR_INPUT
	Prio					: DINT; 					(*1=highest, .. , 4=lowest*)
	Btn1Addr 			: POINTER TO BOOL;	(*Address of Button1 , if Zero then Button is unvisible*)
	Btn2Addr 			: POINTER TO BOOL;	(*Address of Button2 , if Zero then Button is unvisible*)
	Msg				: sMessageText;
	MessageLine		: ARRAY [1..10] OF sMessageLine;
	MsgButton1Text		: STRING(20);
	MsgButton2Text		: STRING(20);

	FB_ReadXmlLineMsg	:FB_ReadXmlLine;
END_VAR
VAR_IN_OUT
	sVisu				: sMessageVisu;
END_VAR
VAR_OUTPUT
	MessageActive		: BOOL;
END_VAR
VAR
	EmptyMsg			: sMessageText;
	TempMsg			: sMessageText;
	TempPrio			: DINT;
	MessageGoneFlag	: F_TRIG;
	MessageShowFlag	: R_TRIG;
	Idx, i					: DINT;
	BackupVisu			: STRING;
	ShowVisuMessage	: BOOL;
	VisuMessageActivT	: TON;

	Button1				: VisuButton;
	Button2				: VisuButton;
	btnHide				: VisuButton;
	btnShow			: VisuButton;
	ShowText			: STRING(255);
	LaufschriftShowText	: FB_Laufschrift_STR255;

(* Vars for Disabling Multiselection *)
	Index			: DINT;
	Index_Clear			: DINT;
	FP_MsgLineBool	: ARRAY[1..20] OF R_TRIG;
	LastPressedLine		: DINT;

	Error				: ErrorStruct;
	ErrorPuls			: BOOL:=FALSE;

END_VAR
(*Das ist noch Baustelle!
Es gibt 2 Möglichkeiten:
a) Prio bei Messages mit Button gibt es nicht.
   Wenn eine Meldung mit Button angezeigt wird, dann solange bis diese quittiert ist.
   Dann erst kommt die nächste dran.

b) Jede Meldung mit Button erhält eine eindeutige PLCID.
   Die Visu schreibt für die angezeigte Meldung die ID zurück in VisuID.
   Wenn das Button-Signal in der PLC ankommt werden die IDs verglichen,
   und nur bei VisuID=PLCID wird der Button an die Aufrufstelle weitergereicht.
*)

Lng();

IF 	(NOT TempMsg.ShowMessage OR
	 Msg.Name=TempMsg.Name AND Msg.Text=TempMsg.Text) THEN
	IF 	Msg.Name=TempMsg.Name	AND
		Msg.Text=TempMsg.Text THEN
		IF 	Btn1Addr<>0 THEN
			IF 	MsgButton1Text='' THEN
				MsgButton1Text:='OK';
			END_IF
			Button1.Enable:=TRUE;
			Button1.Visible:=TRUE;
			Button1.TextOn:=MsgButton1Text;
			IF 	sVisu.Button1.Pressed THEN
				Btn1Addr^:=TRUE;
				MessageLine:=sVisu.MessageLine;
				TempMsg.ShowMessage:=FALSE;
			END_IF
		ELSE
			Button1.Visible:=FALSE;
		END_IF

		IF 	Btn2Addr<>0 THEN
			IF 	MsgButton2Text='' THEN
				MsgButton2Text:='Cancel';
			END_IF
			Button2.Enable:=TRUE;
			Button2.Visible:=TRUE;
			Button2.TextOn:=MsgButton2Text;
			IF 	sVisu.Button2.Pressed THEN
				Btn2Addr^:=TRUE;
				TempMsg.ShowMessage:=FALSE;
			END_IF
		ELSE
			Button2.Visible:=FALSE;
		END_IF
	ELSE
		TempMsg:=Msg;
		sVisu.MessageLine:=MessageLine;
	END_IF
	TempMsg.ShowMessage:=TRUE;
	TempPrio:=Prio;

	IF 	NOT ErrorPuls OR
		Error.DateTime = ErrorHandler.EmptyError.DateTime THEN
		Error.DateTime	:= gVarDTSystemtime;
		ErrorPuls 		:= TRUE;
	END_IF
	Error.Text	:= CONCAT('MessageHandler: ',Msg.Text);
	Error.No		:= 1;
	Error.Typ	:= 1;			(* 0=red 1:=orange 2:=blue *)

	IF 	Error.Text<>'' AND
		ST_Lng.b_EndChangeLng THEN
		ErrorHandler.AddError(	ErrorToAdd:=Error,
								sVisu:=Visu.ErrorHandler);
	END_IF
END_IF


(*Clear Input-Var*)
Prio:=0;
Btn1Addr:=0;
Btn2Addr:=0;
Msg:=EmptyMsg;
MsgButton1Text:='';
MsgButton2Text:='';
END_PROGRAM
ACTION ClearAll:
IF NOT sVisu.ShowMessage THEN
	TempPrio:=0;
	TempMsg.Name:='';
	TempMsg.Text:='';
	TempMsg.ID:='';
	TempMsg.ShowMessage:=FALSE;
	TempMsg.Color:=0;
	TempMsg.Station:=0;
	TempMsg.Button1.Visible:=FALSE;
	TempMsg.Button2.Visible:=FALSE;
ELSE
	TempMsg.ShowMessage:=FALSE;
END_IF

(* Copy from visu *)
MessageLine:=sVisu.MessageLine;
END_ACTION
ACTION ClearMessageLines:
FOR idx:=1 TO 10 DO
	MessageHandler.MessageLine[idx].Visible:=FALSE;
	MessageHandler.MessageLine[idx].Editable:=FALSE;
	MessageHandler.MessageLine[idx].Text:='';
	MessageHandler.MessageLine[idx].MsgInt:=0;
	MessageHandler.MessageLine[idx].MsgBool:=FALSE;
	MessageHandler.MessageLine[idx].MsgReal:=0.0;
	MessageHandler.MessageLine[idx].MsgString:='';
	MessageHandler.MessageLine[idx].MsgTypeEnum:=MsgDataTypeNone;
END_FOR
END_ACTION
ACTION DisableMultiSelect:
LastPressedLine:=0;

FOR Index:=1 TO 10 DO
	FP_MsgLineBool[Index](CLK:=sVisu.MessageLine[Index].MsgBool);
	IF FP_MsgLineBool[Index].Q THEN
		LastPressedLine:=Index;
		EXIT;
	END_IF
END_FOR

IF LastPressedLine>0 THEN

	FOR Index_Clear:=1 TO 10 DO
		MessageLine[Index_Clear].MsgBool:=(LastPressedLine=Index_Clear);
	END_FOR

END_IF
END_ACTION
ACTION Lng:
IF	TempMsg.ID <> '' THEN

	FB_ReadXmlLineMsg(
		Prefix:= 'MSG',
		ID:= TempMsg.ID,
		File:= 'MSG.xml',
		Text=>);

	IF 	FB_ReadXmlLineMsg.Text <> ''  THEN
		TempMsg.Text:=CONCAT(TempMsg.ID,':$N$R');
		TempMsg.Text:=CONCAT(TempMsg.Text,FB_ReadXmlLineMsg.Text);
		Msg.Text:=TempMsg.Text;

		ShowText:=CONCAT(TempMsg.ID,': ');
		ShowText:=CONCAT(ShowText,FB_ReadXmlLineMsg.Text);
		FOR i:=1 TO 10 DO
			IF	FIND(ShowText, '$N') > 0 THEN
				ShowText:=DELETE (ShowText,1,FIND(ShowText, '$N'));
			END_IF
			IF	FIND(ShowText, '$R') > 0 THEN
				ShowText:=DELETE (ShowText,1,FIND(ShowText, '$R'));
			END_IF
		END_FOR
		IF LEN(ShowText) > 60 THEN
			ShowText:=CONCAT(ShowText,' ->   ');
		END_IF
		LaufschriftShowText(
				N:= 60,
				StepWidth:=1,
				PT:= t#100ms ,
				Text:= ShowText,
				Display=>BtnShow.TextOn
				);
	ELSE
		TempMsg.Text:=CONCAT(TempMsg.ID,':..... ');
	END_IF
ELSE
	ShowText:=TempMsg.Text;
	FOR i:=1 TO 10 DO
		IF	FIND(ShowText, '$N') > 0 THEN
			ShowText:=DELETE (ShowText,1,FIND(ShowText, '$N'));
		END_IF
		IF	FIND(ShowText, '$R') > 0 THEN
			ShowText:=DELETE (ShowText,1,FIND(ShowText, '$R'));
		END_IF
	END_FOR
	IF LEN(ShowText) > 60 THEN
		ShowText:=CONCAT(ShowText,' ->   ');
	END_IF
	LaufschriftShowText(
			N:= 60,
			StepWidth:=1,
			PT:= t#100ms ,
			Text:= ShowText,
			Display=>BtnShow.TextOn
			);
END_IF
END_ACTION
ACTION VisuUpdate:
sVisu.Name:=TempMsg.Name;
sVisu.Text:=TempMsg.Text;
sVisu.ID:=TempMsg.ID;
sVisu.ShowMessage:=TempMsg.ShowMessage;
sVisu.Color:=TempMsg.Color;
sVisu.Station:=TempMsg.Station;

sVisu.Button1:=TempMsg.Button1;
sVisu.Button2:=TempMsg.Button2;


(* Write to visu *)

sVisu.MessageLine:=MessageLine;
FOR idx:=1 TO 10 DO
	CASE sVisu.MessageLine[idx].MsgTypeEnum OF
		MsgDataTypeBool: sVisu.MessageLine[idx].MsgType:='BOOL';
		MsgDataTypeDint: sVisu.MessageLine[idx].MsgType:='DINT';
		MsgDataTypeReal: sVisu.MessageLine[idx].MsgType:='REAL';
		MsgDataTypeString: sVisu.MessageLine[idx].MsgType:='STRING';
	ELSE
		sVisu.MessageLine[idx].MsgType:='';
	END_CASE
END_FOR

MessageGoneFlag(CLK:=sVisu.ShowMessage);
MessageShowFlag(CLK:=sVisu.ShowMessage AND NOT sVisu.BtnShow.Pressed);

(*Meldefenster öffnen, wenn Meldung neu aktiv wird (als Impuls)*)
IF MessageShowFlag.Q AND CurrentVisu<>'ZLIB_VISUMESSAGEHANDLER' THEN
	ShowVisuMessage:=TRUE;
	BackupVisu:=CurrentVisu;
END_IF
VisuMessageActivT(IN:=CurrentVisu='ZLIB_VISUMESSAGEHANDLER' ,PT:=T#1s);
IF 	CurrentVisu='ZLIB_VISUMESSAGEHANDLER'AND
	ShowVisuMessage THEN
	ShowVisuMessage:=FALSE;
END_IF
IF 	ShowVisuMessage THEN
	CurrentVisu:='ZLIB_VISUMESSAGEHANDLER';
END_IF

(*Button "Meldung einblenden" anzeigen, wenn Meldung aktiv aber Meldefenster nicht offen*)
IF 	sVisu.ShowMessage AND
	CurrentVisu<>'ZLIB_VISUMESSAGEHANDLER' AND
	NOT ShowVisuMessage THEN
	BtnShow.Visible:=TRUE;
	BtnShow.Enable:=TRUE;
	BtnShow.ButtBackColor:=Visu.Message.Color;
ELSE
	BtnShow.Visible:=FALSE;
END_IF

(*Button "Minimieren" einblenden, wenn Meldefenster offen*)
IF 	CurrentVisu='ZLIB_VISUMESSAGEHANDLER' THEN
	BtnHide.Visible:=TRUE;
	BtnHide.Enable:=TRUE;
	BtnHide.TextOn:='Meldung minimieren';
	BtnHide.ButtBackColor:=Color.control;
ELSE
	BtnHide.Visible:=FALSE;
END_IF

(*Meldefenster komplett schliessen, wenn keine Meldung mehr ansteht*)
IF 	MessageGoneFlag.Q OR
	BtnHide.Pressed THEN
	IF 	BackupVisu<>'' OR
		BackupVisu='ZLIBVISUMESSAGEHANDLER'THEN
		CurrentVisu:=BackupVisu;
	ELSE
		CurrentVisu:='MAIN';
	END_IF
END_IF;

MessageActive := sVisu.ShowMessage OR sVisu.BtnShow.Visible;


(*VisuButton Handler Call*)
Button1(	Button:= TempMsg.Button1);
Button2(	Button:= TempMsg.Button2);
btnHide(	Button:= sVisu.btnHide);
btnShow(	Button:= sVisu.btnShow);
END_ACTION

(* POU zLibrary/ept/Sprache/FB_ReadXmlLine, ST *)
FUNCTION_BLOCK FB_ReadXmlLine
VAR_INPUT
	Prefix					: STRING;
	ID						: STRING;
	File						: STRING;
END_VAR
VAR_OUTPUT
	Text					: STRING(255);
END_VAR

VAR
	bError							: BOOL;
	nErrId							: UDINT;

	fb_state_entry					: ST_StateEntry;

	CURRENTLANGUAGECopy			: STRING(5);
	IdCopy							: STRING;
END_VAR
(*======================================================
   ST: FB_ReadXmlLine
 ------------------------------------------------------
   Auth: 	Werner Frield    						 
   Date: 	23.12.2020    						     
   Rev.: 		1.0	
   Desc	
	-	Mit diesem FB kann Srachabängig ein Text aus einer xml Datei ausgelesen werden		
	-	Das Programm ST_ReadXmlLine wird zum auslesen benutzt.
	-	Die XML Datei muss im PLC Verzeichnis unter TRANS abgelegt werden und 
		mit der Excel Datei (_Texte.xlsm) erstellt werden.
	-	abhängig von der CURRENTLANGUAGE werden Srachabängig die Texte ausgelesen

Beispiel:
FB_ReadXmlLineConf(
	Prefix:= 'CONFIG',			(*erste Spalte der Excel Datei*)
	ID:= 'ST03_473_B70_0',		(*zweite Spalte der Excel Datei*)
	File:= 'CONFIG.xml',		(* xml Datei Name*)
	Text=> );					(* hier kommt der passende Text zurück. abhängig von der angewählten Sprache (DE, EN,CZ*)

 ========================================================*)
fb_state_entry(i16_pos:= 1);
CASE fb_state_entry.i16_step OF
(*=======================================================*)
INIT_OBJ:

	(*-----------------------Weiterschaltbedingungen----------------------------*)
	fb_state_entry.i16_next_step:=INIT;

(*=======================================================*)
INIT:
	IF	TD.ArtNo <> '' AND CURRENTLANGUAGE <> '' THEN
		fb_state_entry.i16_next_step:=BEREIT;
	END_IF

(*=======================================================*)
BEREIT:	fb_state_entry.s_debugtext:='warte auf Start';

	IF	fb_state_entry.E THEN
		bError:=FALSE;
		IdCopy:= ID;
	END_IF
	IF	Prefix <> '' AND ID <> '' AND
		ST_ReadXmlLine.b_ready THEN

		IF	CURRENTLANGUAGECopy <> CURRENTLANGUAGE OR
			IdCopy <> ID THEN
			IF	Prefix <> 'MSG' THEN
				fb_state_entry.i16_next_step:=110;		(*ST_ReadXmlLine*)
			ELSE
				fb_state_entry.i16_next_step:=210;		(*ST_ReadXmlLineMsg*)
			END_IF
		END_IF
	END_IF

	IF	fb_state_entry.X THEN
		CURRENTLANGUAGECopy := CURRENTLANGUAGE;
		Text:='';
	END_IF

(*=======================================================*)
110:  fb_state_entry.s_debugtext:='*Warten bis Lesen erlaubt ist';

	IF	TestAndSet(ST_ReadXmlLine.LockFlag) THEN
		fb_state_entry.i16_next_step := 120;
	END_IF

	IF	fb_state_entry.X THEN
		ST_ReadXmlLine.b_start:=TRUE;
		ST_ReadXmlLine.s_Prefix:= Prefix;
		ST_ReadXmlLine.s_ID:= ID;
		ST_ReadXmlLine.s_File:= File;
		ST_ReadXmlLine.s_Text;
	END_IF

(*=======================================================*)
120:  fb_state_entry.s_debugtext:='*Warten auf busy';

	IF 	ST_ReadXmlLine.b_busy THEN
		fb_state_entry.i16_next_step := 130;
	ELSIF
		fb_state_entry.fb_ton_Step.ET > t#3000ms THEN
		nErrId := ST_ReadXmlLine.nErrId;
		fb_state_entry.s_debugtext:='timeout';
		fb_state_entry.i16_next_step := FEHLER;
	END_IF

(*=======================================================*)
130:  fb_state_entry.s_debugtext:='*Warten auf fertig';

	IF 	ST_ReadXmlLine.b_done THEN
		text:=ST_ReadXmlLine.s_Text;

		fb_state_entry.i16_next_step := BEREIT;
	ELSIF
		fb_state_entry.fb_ton_Step.ET > t#3000ms THEN
		nErrId := ST_ReadXmlLine.nErrId;
		fb_state_entry.s_debugtext:='timeout';
		fb_state_entry.i16_next_step := FEHLER;
	END_IF

(*=======================================================*)
(*=======================================================*)
210:  fb_state_entry.s_debugtext:='*Warten bis Lesen erlaubt ist';

	IF	TestAndSet(ST_ReadXmlLineMsg.LockFlag) THEN
		fb_state_entry.i16_next_step := 220;
	END_IF

	IF	fb_state_entry.X THEN
		ST_ReadXmlLineMsg.b_start:=TRUE;
		ST_ReadXmlLineMsg.s_Prefix:= Prefix;
		ST_ReadXmlLineMsg.s_ID:= ID;
		ST_ReadXmlLineMsg.s_File:= File;
		ST_ReadXmlLineMsg.s_Text;
	END_IF

(*=======================================================*)
220:  fb_state_entry.s_debugtext:='*Warten auf busy';

	IF 	ST_ReadXmlLineMsg.b_busy THEN
		fb_state_entry.i16_next_step := 230;
	ELSIF
		fb_state_entry.fb_ton_Step.ET > t#3000ms THEN
		nErrId := ST_ReadXmlLineMsg.nErrId;
		fb_state_entry.s_debugtext:='timeout';
		fb_state_entry.i16_next_step := FEHLER;
	END_IF

(*=======================================================*)
230:  fb_state_entry.s_debugtext:='*Warten auf fertig';

	IF 	ST_ReadXmlLineMsg.b_done THEN
		text:=ST_ReadXmlLineMsg.s_Text;
		fb_state_entry.i16_next_step := BEREIT;
	ELSIF
		fb_state_entry.fb_ton_Step.ET > t#3000ms THEN
		nErrId := ST_ReadXmlLineMsg.nErrId;
		fb_state_entry.s_debugtext:='timeout';
		fb_state_entry.i16_next_step := FEHLER;
	END_IF

(*=======================================================*)
FEHLER:
	IF 	fb_state_entry.E THEN
		bError:=TRUE;
		Text:=ST_ReadXmlLine.s_Text;
	END_IF

	fb_state_entry.s_debugtext:='nErrorID: ';
	fb_state_entry.s_debugtext:=CONCAT(fb_state_entry.s_debugtext, UDINT_TO_STRING(nErrId));
	fb_state_entry.i16_next_step:=BEREIT;

END_CASE
fb_state_entry(i16_pos:= 2);
END_FUNCTION_BLOCK

(* POU zLibrary/ept/Funktionsbausteine/ST_StateEntry, ST *)
FUNCTION_BLOCK ST_StateEntry
VAR
	arr_last_step_history	: ARRAY[0..31] OF STRING(110);
	last_pos 			: INT := 0;
	interner_step		: INT := 0;
	s_stepTime 			: STRING;
END_VAR
VAR_OUTPUT
	i16_last_step 			: enum_step_nr := INIT_OBJ;	(* Der Schritt vor diesem Schritt *)
	i16_step 				: enum_step_nr := INIT_OBJ;	(* Diese variable soll vom "case step of" verwendet werden *)
	E					: BOOL;					(* Aktiv bei betreten des Steps *)
	X					: BOOL;					(* Aktiv beim verlassen des Steps *)
	b_error 				: BOOL := FALSE;			(* Ablauf Pos 1,2,1,2,1,2,... nicht richtig *)
	fb_ton_Step			: TON;
END_VAR
VAR_INPUT
	i16_next_step 		: enum_step_nr := INIT_OBJ;	(* Nächster schritt *)
	i16_pos 				: INT;					(* Pos = 1: Aufruf vor dem Case step of ---  Pos = 2: Aufruf nach dem Case step of*)
	s_debugtext			: STRING(100);
END_VAR
VAR_TEMP
	i					: INT := 0;
END_VAR
VAR CONSTANT
	t_MaxStepTime		: TIME := T#60S;
END_VAR
(*stepTime ermitteln*)
fb_ton_Step(IN:= , PT:=fb_ton_Step.ET + t#10s , Q=>  , ET=> );
IF	i16_step = i16_next_step THEN
	fb_ton_Step.IN:=TRUE;
END_IF

IF	NOT b_error THEN
	CASE interner_step OF
		0:
			(* Mitten im Schritt drin *)
			X := FALSE;
			E := FALSE;


			(* Schritt wird verlassen *)
			IF i16_step <> i16_next_step AND i16_pos = 1 THEN
				subrDebugtext();
				interner_step := 10;
				X := TRUE;
				E := FALSE;
				fb_ton_Step.IN:=FALSE;
			END_IF

		10:
			(* Eintritt in neuen Schritt *)
			IF i16_pos = 1 THEN
				X := FALSE;
				E := TRUE;

				(* Schalte Schritt weiter *)
				i16_last_step := i16_step;
				i16_step := i16_next_step;
				(* Baue Statehistory *)

				IF  E THEN
					FOR i:= 31 TO 1 BY -1 DO
						arr_last_step_history[i] := arr_last_step_history[i-1];
					END_FOR
					arr_last_step_history[0] := '';
					s_stepTime:='';
					s_debugtext:='';
				END_IF

				interner_step := 0;

			END_IF
	END_CASE
END_IF

IF 	(fb_ton_Step.ET >= T#200ms AND arr_last_step_history[0] = '') OR	(* Am Anfang Debugtext schreiben, damit etwas drin steht *)
	(fb_ton_Step.Q AND s_stepTime <> '>1m') THEN	(* Debugtext schreiben, wenn t_MaxStepTime erreicht wird *)
	subrDebugtext();
END_IF

(* Prüfe Baustein *)
IF 	i16_pos = last_pos THEN
	b_error := TRUE;
END_IF

last_pos := i16_pos;
END_FUNCTION_BLOCK
ACTION subrDebugtext:
s_stepTime:=ET_TO_STRING(fb_ton_Step.ET);
IF 	fb_ton_Step.ET >= t_MaxStepTime THEN
	s_stepTime:=CONCAT('>',s_StepTime);
END_IF

(* history zusammenbauen aus StepNr, StepTime und debugtext*)
CASE i16_step OF
	INIT_OBJ :			arr_last_step_history[0]:='INIT_OBJ';
	INIT :				arr_last_step_history[0]:='INIT';
	BEREIT :			arr_last_step_history[0]:='BEREIT';
	HALT :				arr_last_step_history[0]:='HALT';
	STOP :				arr_last_step_history[0]:='STOP';
	FEHLER :			arr_last_step_history[0]:='FEHLER';
	INAKTIV:			arr_last_step_history[0]:='INAKTIV ';
ELSE
	arr_last_step_history[0] := INT_TO_STRING(i16_step);
END_CASE

IF 	s_stepTime ='0ms' OR s_stepTime =''THEN
	s_stepTime:='3ms';		(*damit nicht 0 drin steht*)
END_IF
arr_last_step_history[0] := CONCAT(arr_last_step_history[0],':  ');
arr_last_step_history[0] := CONCAT(arr_last_step_history[0],s_stepTime);
arr_last_step_history[0] := CONCAT(arr_last_step_history[0],': ');
arr_last_step_history[0] := CONCAT(arr_last_step_history[0],s_debugtext);
END_ACTION

(* POU zLibrary/ept/Funktionen/ET_TO_STRING, ST *)
FUNCTION ET_TO_STRING :STRING
VAR_INPUT
	et		:TIME;
END_VAR

VAR

END_VAR
ET_TO_STRING:=TIME_TO_STRING(et);
ET_TO_STRING:=DELETE(ET_TO_STRING,2,1);
END_FUNCTION

(* POU zLibrary/ept/Sprache/ST_ReadXmlLine, ST *)
PROGRAM ST_ReadXmlLine (*Programm wird nur vom FB_ReadXmlLine benutzt*)
VAR_INPUT
	b_start					: BOOL;
	s_Prefix					: STRING;
	s_ID					: STRING;
	s_File					: STRING;
	s_XmlHelp				: T_MaxString;	(* in diese Variable schreibt der XML-Bautstein die ausgelesenen Daten *)
END_VAR
VAR_OUTPUT
	b_EndChangeLng		: BOOL;
	b_busy					: BOOL;
	b_ready					: BOOL;
	b_done					: BOOL;

	s_Text					: STRING(255);
END_VAR

VAR

	LockFlag						: BOOL := FALSE;	(* Ganz wichtig, wenn diese Variable TRUE ist, dann kann die Struktur "Visu.MeldungProduktion" nicht verändert werden *)
	b_Error							: BOOL;
	nErrId							: UDINT;
	s_filePath						: T_MaxString;
	s_Xpath							: T_MaxString;

	fb_state_entry					: ST_StateEntry;
	fb_xml_srv_read					: FB_XmlSrvReadByName;	(* XML Baustein zum Auslesen der CONFIG *)

	CURRENTLANGUAGECopy			: STRING(5);
END_VAR
VAR CONSTANT
	s_SymName					: STRING:='ST_ReadXmlLine.s_XmlHelp';
END_VAR
(*Programm wird nur vom FB_ReadXmlLine benutzt*)

(*===================================================================================================*)
fb_state_entry(i16_pos:= 1);

CASE fb_state_entry.i16_step OF
(*=======================================================*)
INIT_OBJ:

	fb_state_entry.i16_next_step:=INIT;

(*=======================================================*)
INIT:

	IF	TD.ArtNo <> '' THEN
		fb_state_entry.i16_next_step:=BEREIT;
	END_IF

(*=======================================================*)
BEREIT:	fb_state_entry.s_debugtext:='warte auf Start';

	IF	fb_state_entry.E THEN
		b_Error:=FALSE;
		b_ready:=TRUE;
		LockFree();
	END_IF

	IF	s_Prefix <> '' AND s_ID <> '' AND
		b_start THEN
		fb_state_entry.i16_next_step:=110;
(*		LockGet();	(* Ablauf ist immer derselbe, zuerst LockGet, dann Strukturen ändern, dann LockFree *)*)
	END_IF

	IF	fb_state_entry.fb_ton_Step.ET >t#10ms THEN
		b_EndChangeLng:=TRUE;
	END_IF

	IF	fb_state_entry.X THEN
		IF 	CURRENTLANGUAGECopy<>CURRENTLANGUAGE THEN
			CURRENTLANGUAGECopy:=CURRENTLANGUAGE;
			b_EndChangeLng:=FALSE;
		END_IF
		s_XmlHelp:='';
		s_Text:='';
		b_ready:=FALSE;
		b_done:=FALSE;
		b_busy:=TRUE;
	END_IF

(*=======================================================*)
110:	fb_state_entry.s_debugtext:='Zeile aus der XMl auslesen';

	IF	fb_state_entry.E THEN
		s_filePath := CONCAT(s_PLC_path,'TRANS\');
		s_filePath := CONCAT(s_filePath,s_File);

		s_Xpath:= '/dynamic-text/text-list/text[@prefix=$'';
		s_Xpath:=CONCAT(s_Xpath,s_Prefix);
		s_Xpath:=CONCAT(s_Xpath,'$' and @id=$'');
		s_Xpath:=CONCAT(s_Xpath,s_ID);
		s_Xpath:=CONCAT(s_Xpath,'$']/');
		s_Xpath:=CONCAT(s_Xpath, CURRENTLANGUAGE);
	END_IF

	(*-----------------------Weiterschaltbedingungen----------------------------*)
	fb_state_entry.i16_next_step := 120;

(*=======================================================*)
120:	fb_state_entry.s_debugtext:='Starte Daten lesen ';

	IF 	fb_state_entry.E THEN
		fb_xml_srv_read.sFilePath := s_filePath;
		fb_xml_srv_read.sXPath :=s_Xpath;
		fb_xml_srv_read.sSymName := s_SymName;
		fb_xml_srv_read.bExecute := TRUE;
	END_IF

	(*-----------------------Weiterschaltbedingungen----------------------------*)
	IF 	fb_xml_srv_read.bBusy THEN
		fb_xml_srv_read.bExecute := FALSE;
		fb_state_entry.i16_next_step := 130;
	END_IF

(*=======================================================*)
130:fb_state_entry.s_debugtext:='warte auf fertig';

	(*-----------------------Weiterschaltbedingungen----------------------------*)
	IF  	NOT fb_xml_srv_read.bBusy  THEN
		fb_state_entry.i16_next_step := 140;
	ELSIF
		fb_state_entry.fb_ton_Step.ET > t#3000ms THEN
		nErrId := fb_xml_srv_read.nErrId;
		fb_state_entry.s_debugtext:='timeout';
		fb_state_entry.i16_next_step := FEHLER;
	END_IF

(*=======================================================*)
140:fb_state_entry.s_debugtext:='prüfe auf Fehler';

	(*-----------------------Weiterschaltbedingungen----------------------------*)
	IF  	fb_xml_srv_read.bError OR
		s_XmlHelp = '' THEN
		nErrId := fb_xml_srv_read.nErrId;
		fb_state_entry.i16_next_step := FEHLER;
	ELSE
		s_Text:=s_XmlHelp;
		fb_state_entry.i16_next_step := BEREIT;
		b_done:=TRUE;
		b_busy:=FALSE;
	END_IF


(*=======================================================*)
FEHLER:
	IF 	fb_state_entry.E THEN
		b_Error:=TRUE;
		s_Text:='!!! ';
		s_Text:= CONCAT(s_Text,s_Prefix);
		s_Text:= CONCAT(s_Text,'-');
		s_Text:= CONCAT(s_Text,s_ID);
		s_Text:= CONCAT(s_Text,' not found !!!');
	END_IF

	fb_state_entry.s_debugtext:='nErrorID: ';
	fb_state_entry.s_debugtext:=CONCAT(fb_state_entry.s_debugtext, UDINT_TO_STRING(nErrId));
	fb_state_entry.s_debugtext:=CONCAT(fb_state_entry.s_debugtext, ' =>');
	fb_state_entry.s_debugtext:=CONCAT(fb_state_entry.s_debugtext, s_Text);

	(*-----------------------Weiterschaltbedingungen----------------------------*)
	fb_state_entry.i16_next_step:=BEREIT;

	IF 	fb_state_entry.E THEN
		b_done:=TRUE;
		b_busy:=FALSE;
	END_IF

END_CASE

fb_state_entry(i16_pos:= 2);

b_start:=FALSE;


(* XML *)
fb_xml_srv_read(
	sNetId:= '',
	ePath:= PATH_GENERIC,
	nMode:= XMLSRV_SKIPMISSING,
	sSymName:= ,
	sFilePath:= ,
	sXPath:= ,
	bExecute:= ,
	tTimeout:= t#10s,
	bBusy=> ,
	bError=> ,
	nErrId=> );
END_PROGRAM
ACTION LockFree:
LockFlag := FALSE;	(* wieder freigeben *)
END_ACTION
ACTION LockGet:
WHILE NOT TestAndSet(LockFlag) DO	(* Mit der Funktion TestAndSet kann ein Flag nicht unterbrechbar geprüft und gesetzt werden *)
	;	(* Wait until Lock is free *)
END_WHILE
(*LockFlag: Ist ein boolsches Flag, das geprüft wird
 - war es FALSE, dann war das Flag frei und wird gesetzt (blockiert von nun an), die Funktion liefert TRUE
 - war es TRUE, dann war das Flag bereits belegt (blockiert), die Funktion liefert FALSE*)
END_ACTION

(* POU zLibrary/ept/Sprache/ST_ReadXmlLineMsg, ST *)
PROGRAM ST_ReadXmlLineMsg
VAR_INPUT
	b_start					: BOOL;
	s_Prefix					: STRING;
	s_ID					: STRING;
	s_File					: STRING;
	s_XmlHelp				: T_MaxString;	(* in diese Variable schreibt der XML-Bautstein die ausgelesenen Daten *)
END_VAR
VAR_OUTPUT
	b_EndChangeLng		: BOOL;
	b_busy					: BOOL;
	b_ready					: BOOL;
	b_done					: BOOL;

	s_Text					: STRING(255);
END_VAR

VAR
	LockFlag						: BOOL := FALSE;	(* Ganz wichtig, wenn diese Variable TRUE ist, dann kann die Struktur "Visu.MeldungProduktion" nicht verändert werden *)
	b_Error							: BOOL;
	nErrId							: UDINT;
	s_filePath						: T_MaxString;
	s_Xpath							: T_MaxString;

	fb_state_entry					: ST_StateEntry;
	fb_xml_srv_read					: FB_XmlSrvReadByName;	(* XML Baustein zum Auslesen der CONFIG *)

	CURRENTLANGUAGECopy			: STRING(5);
END_VAR
VAR CONSTANT
	s_SymName					: STRING:='ST_ReadXmlLineMsg.s_XmlHelp';
END_VAR
(*===================================================================================================*)
fb_state_entry(i16_pos:= 1);

CASE fb_state_entry.i16_step OF
(*=======================================================*)
INIT_OBJ:

	fb_state_entry.i16_next_step:=INIT;

(*=======================================================*)
INIT:

	IF	TD.ArtNo <> '' THEN
		fb_state_entry.i16_next_step:=BEREIT;
	END_IF

(*=======================================================*)
BEREIT:	fb_state_entry.s_debugtext:='warte auf Start';

	IF	fb_state_entry.E THEN
		b_Error:=FALSE;
		b_ready:=TRUE;
		LockFree();
	END_IF

	IF	s_Prefix <> '' AND s_ID <> '' AND
		b_start THEN
		fb_state_entry.i16_next_step:=110;
(*		LockGet();	(* Ablauf ist immer derselbe, zuerst LockGet, dann Strukturen ändern, dann LockFree *)*)
	END_IF

	IF	fb_state_entry.fb_ton_Step.ET >t#10ms THEN
		b_EndChangeLng:=TRUE;
	END_IF

	IF	fb_state_entry.X THEN
		IF 	CURRENTLANGUAGECopy<>CURRENTLANGUAGE THEN
			CURRENTLANGUAGECopy:=CURRENTLANGUAGE;
			b_EndChangeLng:=FALSE;
		END_IF
		s_XmlHelp:='';
		s_Text:='';
		b_ready:=FALSE;
		b_done:=FALSE;
		b_busy:=TRUE;
	END_IF

(*=======================================================*)
110:	fb_state_entry.s_debugtext:='Zeile aus der XML auslesen';

	IF	fb_state_entry.E THEN
		s_filePath := CONCAT(s_PLC_path,'TRANS\');
		s_filePath := CONCAT(s_filePath,s_File);

		s_Xpath:= '/dynamic-text/text-list/text[@prefix=$'';
		s_Xpath:=CONCAT(s_Xpath,s_Prefix);
		s_Xpath:=CONCAT(s_Xpath,'$' and @id=$'');
		s_Xpath:=CONCAT(s_Xpath,s_ID);
		s_Xpath:=CONCAT(s_Xpath,'$']/');
		s_Xpath:=CONCAT(s_Xpath, CURRENTLANGUAGE);
	END_IF

	(*-----------------------Weiterschaltbedingungen----------------------------*)
	fb_state_entry.i16_next_step := 120;

(*=======================================================*)
120:	fb_state_entry.s_debugtext:='Starte Daten lesen ';

	IF fb_state_entry.E THEN
		fb_xml_srv_read.sFilePath := s_filePath;
		fb_xml_srv_read.sXPath :=s_Xpath;
		fb_xml_srv_read.sSymName := s_SymName;
		fb_xml_srv_read.bExecute := TRUE;
	END_IF

	(*-----------------------Weiterschaltbedingungen----------------------------*)
	IF 	fb_xml_srv_read.bBusy THEN
		fb_xml_srv_read.bExecute := FALSE;
		fb_state_entry.i16_next_step := 130;
	END_IF

(*=======================================================*)
130:fb_state_entry.s_debugtext:='warte auf fertig';

	(*-----------------------Weiterschaltbedingungen----------------------------*)
	IF  	NOT fb_xml_srv_read.bBusy  THEN
		fb_state_entry.i16_next_step := 140;
	ELSIF
		fb_state_entry.fb_ton_Step.ET > t#3000ms THEN
		nErrId := fb_xml_srv_read.nErrId;
		fb_state_entry.s_debugtext:='timeout';
		fb_state_entry.i16_next_step := FEHLER;
	END_IF

(*=======================================================*)
140:fb_state_entry.s_debugtext:='prüfe auf Fehler';

	(*-----------------------Weiterschaltbedingungen----------------------------*)
	IF  	fb_xml_srv_read.bError OR
		s_XmlHelp = '' THEN
		nErrId := fb_xml_srv_read.nErrId;
		fb_state_entry.i16_next_step := FEHLER;
	ELSE
		s_Text:=s_XmlHelp;
		fb_state_entry.i16_next_step := BEREIT;
		b_done:=TRUE;
		b_busy:=FALSE;
	END_IF


(*=======================================================*)
FEHLER:
	IF 	fb_state_entry.E THEN
		b_Error:=TRUE;
		s_Text:='!!! ';
		s_Text:= CONCAT(s_Text,s_Prefix);
		s_Text:= CONCAT(s_Text,'-');
		s_Text:= CONCAT(s_Text,s_ID);
		s_Text:= CONCAT(s_Text,' not found !!!');
	END_IF

	fb_state_entry.s_debugtext:='nErrorID: ';
	fb_state_entry.s_debugtext:=CONCAT(fb_state_entry.s_debugtext, UDINT_TO_STRING(nErrId));
	fb_state_entry.s_debugtext:=CONCAT(fb_state_entry.s_debugtext, ' =>');
	fb_state_entry.s_debugtext:=CONCAT(fb_state_entry.s_debugtext, s_Text);

	(*-----------------------Weiterschaltbedingungen----------------------------*)
	fb_state_entry.i16_next_step:=BEREIT;

	IF 	fb_state_entry.E THEN
		b_done:=TRUE;
		b_busy:=FALSE;
	END_IF

END_CASE

fb_state_entry(i16_pos:= 2);

b_start:=FALSE;


(* XML *)
fb_xml_srv_read(
	sNetId:= '',
	ePath:= PATH_GENERIC,
	nMode:= XMLSRV_SKIPMISSING,
	sSymName:= ,
	sFilePath:= ,
	sXPath:= ,
	bExecute:= ,
	tTimeout:= t#10s,
	bBusy=> ,
	bError=> ,
	nErrId=> );
END_PROGRAM
ACTION LockFree:
LockFlag := FALSE;	(* wieder freigeben *)
END_ACTION
ACTION LockGet:
WHILE NOT TestAndSet(LockFlag) DO	(* Mit der Funktion TestAndSet kann ein Flag nicht unterbrechbar geprüft und gesetzt werden *)
	;	(* Wait until Lock is free *)
END_WHILE
(*LockFlag: Ist ein boolsches Flag, das geprüft wird
 - war es FALSE, dann war das Flag frei und wird gesetzt (blockiert von nun an), die Funktion liefert TRUE
 - war es TRUE, dann war das Flag bereits belegt (blockiert), die Funktion liefert FALSE*)
END_ACTION

(* POU System/VisuInterface/VisuButton, ST *)
FUNCTION_BLOCK VisuButton
VAR_INPUT
	Enable						:	BOOL := TRUE;
	Visible						:	BOOL := TRUE;
	PressedExt				:	BOOL;
	StateOn						:	BOOL;

	TextColEnabled		:	DINT;
	TextColDisabled		:	DINT;
	ButtColOn					:	DINT;
	ButtBackColor 		:	DINT;
	ButtColDisabled		:	DINT;

	TextOn						:	STRING;
	TextOff						:	STRING(30);

END_VAR
VAR_IN_OUT
	Button				: 	sButtonVisu;

END_VAR

VAR_OUTPUT
	PressedFlag	:	BOOL;
	Pressed			:	BOOL;
END_VAR

VAR
	PressedRTrig	:	R_TRIG;


END_VAR

(* Call of FB
	VisuButton(	Button:=Visu.ButtonAuto,
						Enable:=xxxx  ,
						Visible:=TRUE ,
						PressedExt:=FALSE ,
						StateOn:= xxxx,

						TextColEnabled:= 	Color.black ,
						TextColDisabled:=	Color.white ,
						ButtColOff:= 			Color.grey,
						ButtColOn:= 			Color.lime,
						ButtColPressed:=	Color.yellow ,
						ButtColDisabled:=	Color.lightgrey ,

						TextOn:= 'xxxx',
						TextOff:= 'xxxx',
						);
*)
(* Init colors if not filled *)
 IF 	TextColEnabled = 0 THEN
	TextColEnabled:= 	Color.black ;
END_IF
 IF 	TextColDisabled = 0 THEN
	TextColDisabled:= 	Color.darkgrey ;
END_IF

IF 	ButtBackColor = 0 THEN
	ButtBackColor:= 	Color.control ;
END_IF

IF 	ButtColOn = 0 THEN
	ButtColOn:= 	Color.lime ;
END_IF

IF 	ButtColDisabled = 0 THEN
	ButtColDisabled:= 	Color.control ;
END_IF

(* Check Button pressed *)
Pressed:=Button.Pressed OR PressedExt;

(* Flag button pressed *)
PressedRTrig(CLK:=Pressed);(* AND Enable);*)
PressedFlag:=PressedRTrig.Q;

(* Check button enabled *)
IF 	Enable THEN
	(* Button enabled *)
	Button.TextColor:=TextColEnabled;

	(* Check button pressed *)
	IF 	Pressed THEN
		(* Button pressed *)
		Button.BackgroundColor:=ButtBackColor;
	ELSE
		(* Button not pressed *)

		(* Check state on *)
		IF 	StateOn THEN
			(* State on *)
			Button.BackgroundColor:=ButtColOn;
		ELSE
			(* State off *)
			Button.BackgroundColor:=ButtBackColor;
		END_IF

	END_IF
ELSE
	(* Button not enabled *)
	Button.TextColor:=TextColDisabled;
	Button.Pressed:=FALSE;
	(* Check state on *)
	IF 	StateOn THEN
		(* State on *)
		Button.BackgroundColor:=ButtColOn;
	ELSE
		(* State off *)
		Button.BackgroundColor:=ButtColDisabled;
	END_IF

END_IF

(* Additional assigns to visu *)
Button.Enable:=Enable;
Button.Visible:=Visible;

IF 	StateOn THEN
	(* State on *)
	Button.Text:=TextOn;
ELSE
	(* State off *)
	IF 	TextOff<>'' THEN
		Button.Text:=TextOff;
	ELSE
		Button.Text:=TextOn;
	END_IF
END_IF
END_FUNCTION_BLOCK

(* POU zLibrary/_HelpFunctions/FB_Laufschrift_STR255, ST *)
FUNCTION_BLOCK FB_Laufschrift_STR255
VAR_INPUT
	N 					:INT; (* Max output Stringlength *)
	StepWidth			:INT:=1;
	PT					:TIME;
END_VAR
VAR_IN_OUT
	Text 				:STRING(255); (* Original String *)
END_VAR
VAR_OUTPUT
	Display 				:STRING(255); (* Output String *)
END_VAR
VAR
	delay 				:TP;
	TempOutputString	:STRING(255);
	TempInputText		:STRING(255);
	step 				:INT;
END_VAR
(* generate next ticker when delay is low *)
IF 	N < LEN(text) THEN
	IF 	NOT delay.Q THEN
		(* increase step for next tick *)
		TempInputText:=text;

		step := step + StepWidth;

		IF 	step > LEN(TempInputText) THEN
			step := 1;
		END_IF

		(* extract dispay from text *)
		TempOutputString := MID(TempInputText, N, step);

		IF 	LEN(TempOutputString)<N THEN
			TempOutputString:=CONCAT(TempOutputString,TempInputText);
			TempOutputString:=LEFT(TempOutputString,N);
			Display:=TempOutputString;
		ELSE
			Display:=TempOutputString;
		END_IF
		(* set delay timer for next tick *)
		delay(IN := TRUE, PT := PT);
	ELSE
		(* execute delay timer *)
		delay(IN := FALSE);
	END_IF
ELSE
	display := text;
END_IF
END_FUNCTION_BLOCK

(* POU zLibrary/ept/Sprache/ST_Lng, ST *)
PROGRAM ST_Lng (*Pulldownmenue für Sprachumschaltung*)
VAR_OUTPUT
	b_EndChangeLng		: BOOL;
END_VAR
VAR
	b_init				:BOOL:=FALSE;

	b_einblenden		: BOOL;
	fb_Ton_ChangeLng		: TON;
	fb_ton_ausblenden	: TON;
	fb_rTrig_ausblenden	: R_TRIG;

	s_VisuBmpPath		: STRING(255);
	index				: INT;
	i					: INT;
	CURRENTLANGUAGECopy	: STRING(5);

	btn_Language		:ARRAY [0..5] OF sButtonVisuBmp;

END_VAR
fb_Ton_ChangeLng(
	IN:=	ST_ReadXmlLineMsg.b_EndChangeLng AND
			ST_ReadXmlLine.b_EndChangeLng,
	PT:= t#200ms,
	Q=> b_EndChangeLng,
	ET=> );

IF	NOT b_init THEN
	IF	TD.ArtNo <> '' AND
		s_PLC_path <> '' THEN
		b_init:=TRUE;
		CURRENTLANGUAGE:=MP.ST00.Sprache;
		CURRENTLANGUAGECopy:=CURRENTLANGUAGE;
		s_VisuBmpPath:=CONCAT(s_PLC_path, 'bmp\' );
		Btn_Init();
		IF	CURRENTLANGUAGE ='' THEN
			CURRENTLANGUAGE:='DE';
		END_IF
	END_IF
ELSE
	MP.ST00.Sprache := CURRENTLANGUAGE;
END_IF

ST_Lng.btn_Language[ST_Lng.index].BmpPath;
fb_rTrig_ausblenden(CLK:=b_einblenden);
fb_ton_ausblenden(IN:=, PT:=t#5000ms, Q=>);

IF	fb_rTrig_ausblenden.Q THEN
	fb_ton_ausblenden.IN:=NOT fb_ton_ausblenden.IN;
ELSIF
	fb_ton_ausblenden.Q THEN
	fb_ton_ausblenden.IN:=FALSE;
END_IF

IF  b_init THEN
	FOR i := 0 TO 5  BY 1DO
		IF	CURRENTLANGUAGE=btn_Language[i].Text THEN
			index:=i;
			btn_Language[i].innenFarbe:=Color.darkgrey;
		ELSE
			btn_Language[i].innenFarbe:=Color.lightgrey;
		END_IF

		IF	btn_Language[i].tasten THEN
			CURRENTLANGUAGE:=btn_Language[i].Text;
			fb_ton_ausblenden.IN:=FALSE;
		END_IF
	END_FOR
	CURRENTLANGUAGECopy:=CurrentLanguage;
END_IF
END_PROGRAM
ACTION Btn_Init:
(*=====================================================================*)
btn_Language[0].Text:='DE';
btn_Language[1].Text:='EN';
btn_Language[2].Text:='CZ';
btn_Language[3].Text:='';
btn_Language[4].Text:='';
btn_Language[5].Text:='';

FOR i := 0 TO 5  BY 1DO
	btn_Language[i].deaktivieren:=FALSE;
	btn_Language[i].Textfarbe:=Color.black;
	btn_Language[i].BmpPath:=s_VisuBmpPath;

	btn_Language[i].BmpPath:=CONCAT(btn_Language[i].BmpPath,btn_Language[i].Text);
	btn_Language[i].BmpPath:=CONCAT(btn_Language[i].BmpPath,'.bmp');
	IF	btn_Language[i].Text = '' THEN
		btn_Language[i].unsichtbar:= TRUE;
	ELSE
		btn_Language[i].unsichtbar:= FALSE;
	END_IF

END_FOR
END_ACTION

(* POU System/VisuInterface/ModeSelect, ST *)
PROGRAM ModeSelect (*28.JUL 2010, g.baiz (mit korrigiertem iRemoteAutoStart und iRemoteAutoStop) *)

VAR_OUTPUT
	HomePosition				:	BOOL;
	State								: DINT;
	Mode								:	StateMode;	          (*Betriebsarten / mode*)
	BasicManualMode			:	BOOL	:=	FALSE;
	BasicAutoMode				:	BOOL	:=	FALSE;
	QReset							:	BOOL	:=	FALSE;
	GlobalEnable		:	BOOL	:=	TRUE;
	ControlIsOn			: BOOL;
	ManualFirstImp		: BOOL	:=	FALSE;
	StepFirstImp		: BOOL	:=	FALSE;
	AutoFirstImp		: BOOL	:=	FALSE;
	HomePosRunFirstImp	: BOOL	:=	FALSE;
	QProtecKeyNotIn		: BOOL	:=	FALSE;
	QProtecNotBridged	: BOOL	:=	FALSE;
END_VAR
VAR_INPUT
	(* Inputs from SFC's (used from the application programmer) *)
	AskForNoMode			: BOOL;
	AskForManual			: BOOL;
	AskForStepMode			: BOOL;
	AskForStepStop			: BOOL;
	AskForStepStart			: BOOL;
	AskForAutoMode			: BOOL;
	AskForAutoStart			: BOOL;
	AskAutoStartOverHomePosRun : BOOL;
	AskForAutoStop			: BOOL;
	AskForHomePos			: BOOL;
	AskForSpecialMode		: BOOL;
	(**)
	iRemoteAutoStart		: BOOL;
	iRemoteAutoStop			: BOOL;
	(* Inputs from other FB's (used for call in Special) *)
	ControlOn				: BOOL;
	ProtecKeyNotIn			: BOOL;
	ProtecNotBridged		: BOOL;
	EnableFromPrevMach		: BOOL;
	EnableFromNextMach		: BOOL;
	AllDoorsClosed			: BOOL;
	SafetyDoorOk			: BOOL;
	MainValveOk				: BOOL;
	EmergencyOk				: BOOL;
	BusControlState			: DINT;
	UserOK					: BOOL;
	(* Inputs from MainSequences (signal for Sequence-End) *)
	AutoCycleEnd			: BOOL;
	SpecialCycleEnd 		: BOOL;
	HomePosRunEnd			: BOOL;
	DisableManualMode		: BOOL; 	(* Do not show button for manual mode. This can avoid that automatic cycle is interrupted by operator *)
	RunEmptyEnd				: BOOL; 	(*CellIsEmpty*)
	ShowBtnRunEmpty			: BOOL :=TRUE;

	(*Standard-Inputs *)
	sInit					: sModeSelectInit;(* stuct for initializing*)
											(* Initialisierungsstruktur*)
	Enable					: BOOL; 		(* Enables the operations *)
									 		(* Freigabe für Aktion *)
	Reset					: BOOL; 		(* resetting the Objekt *)
											(* Zurücksetzen des Objektes *)
END_VAR

VAR
	BtnManual		: VisuButton;
	BtnStep			: VisuButton;
	BtnStepCycle	: VisuButton;
	BtnAuto			: VisuButton;
	BtnAutoStart	: VisuButton;
	BtnAutoStop		: VisuButton;
	BtnRunEmpty		: VisuButton;
	BtnHomeRun		: VisuButton;
	BtnSpecial		: VisuButton;
	BtnSpecStep		: VisuButton;
	BtnReset		: VisuButton;

	(* Internal Variables *)
	ErrorNo			: DINT;
	ErrorText		: STRING(80);
	InternNextStep	: BOOL;
	InternResetMode	: DINT;
	InternLastMode	: DINT;
	StepToAuto		: BOOL;
	ShowButton		: BOOL;
	HardwareOk		: BOOL;
	ResetFlag		: R_TRIG;
	ton_Reset		: TON;

	HomePositionInfoNo		: DINT;					(* missing to home posistion /  Fehlernummer fehlende Grundstellung *)
 	NoModeFirstImp			: R_TRIG;
	TipInSpecialMode		: BOOL;
END_VAR
VAR_IN_OUT
	sVisu					: sModeSelectVisu;
END_VAR
VAR CONSTANT
	RESET_FOR_MANUAL			: DINT:=1;
	RESET_FOR_STEP				: DINT:=2;
	RESET_FOR_AUTO				: DINT:=3;
	RESET_FOR_MODE_HOME_POS_RUN	: DINT:=4;
END_VAR
(* Manual mode *)
BtnManual(		Button:=sVisu.BtnManual,
				PressedExt:=FALSE ,
				StateOn:= Mode=MODE_MANUAL ,
				TextOn:='Manual',
				TextOff:='Manual',
				);

(* Step  *)
BtnStep(		Button:=sVisu.BtnStep,
				PressedExt:=FALSE ,
				StateOn:= Mode=MODE_STEP OR Mode=MODE_STEP_RUN,
				TextOn:='Step',
				TextOff:='Step',
				);
(* Step cycle *)
BtnStepCycle(	Button:=sVisu.BtnStepCycle,
				PressedExt:=FALSE ,
				StateOn:= gTipImp ,
				TextOn:='StepCycle',
				TextOff:='StepCycle',
				);
(* Auto mode *)
BtnAuto(		Button:=sVisu.BtnAuto,
				PressedExt:=FALSE ,
				StateOn:= (Mode=MODE_AUTO OR Mode=MODE_AUTO_RUN OR Mode=MODE_AUTO_STOP OR Mode=MODE_HOME_POS_RUN),
				TextOn:='Auto',
				TextOff:='Auto',
				);
(* Auto start *)
BtnAutoStart(	Button:=sVisu.BtnAutoStart,
				PressedExt:=FALSE ,
				StateOn:= Mode=MODE_AUTO_RUN,
				TextOn:='AutoStart',
				TextOff:='AutoStart',
				);
(* Auto stop *)
BtnAutoStop(	Button:=sVisu.BtnAutoStop,
				PressedExt:=FALSE ,
				StateOn:= Mode=MODE_AUTO_STOP,
				TextOn:='AutoStop',
				TextOff:='AutoStop',
				);
(* RunEmpty *)
BtnRunEmpty(	Button:=sVisu.BtnRunEmpty,
				PressedExt:=FALSE ,
				StateOn:=gRunEmpty,
				TextOn:='RunEmpty',
				TextOff:='RunEmpty',
				);
(* SpecialMode *)
BtnSpecial(		Button:=sVisu.BtnSpecial,
				PressedExt:=FALSE ,
				StateOn:= Mode=MODE_SPECIAL,
				TextOn:='Special',
				TextOff:='Special',
				);
(* Step in SpecialMode *)
BtnSpecStep(	Button:=sVisu.BtnSpecStep,
				PressedExt:=FALSE ,
				StateOn:= TipInSpecialMode,
				TextOn:= 'StepCycle',
				TextOff:='StepCycle',
				);
(* Home pos run *)
BtnHomeRun(	Button:=sVisu.BtnHomeRun,
				PressedExt:=FALSE ,
				StateOn:= Mode=MODE_HOME_POS_RUN,
				TextOn:='Home',
				TextOff:='Home',
				);
(*Reset *)
BtnReset(		Button:=sVisu.BtnReset,
				PressedExt:=FALSE ,
				StateOn:= gResetAll,
				TextOn:='Reset',
				TextOff:='Reset',
				);
ManualFirstImp:=FALSE;
StepFirstImp:=FALSE;
AutoFirstImp:=FALSE;
HomePosRunFirstImp:=FALSE;

(*###########################################################################*)
(*    Change Visu Picture																															 *)
(*###########################################################################*)
IF 	BtnAutoStart.PressedFlag THEN
	visu.SelectPictureName:='MAIN';
	CurrentVisu:='MAIN';
END_IF

IF 	BtnHomeRun.PressedFlag THEN
	visu.SelectPictureName:='SYSTEM_GST';
	CurrentVisu:='SYSTEM_GST';
END_IF

(*###########################################################################*)
(* Anwahl von Einzel-, Tipp- oder Automatikbetrieb nach Resetimpuls          *)
(* Select mode																															 *)
(*###########################################################################*)
CASE InternResetMode OF
RESET_FOR_MANUAL:
	Mode:=MODE_MANUAL;
	ManualFirstImp:=TRUE;
RESET_FOR_STEP:
	Mode:=MODE_STEP;
	StepFirstImp:=TRUE;
RESET_FOR_AUTO:
	Mode:=MODE_AUTO;
	AutoFirstImp:=TRUE;
RESET_FOR_MODE_HOME_POS_RUN:
	Mode:=MODE_HOME_POS_RUN;
	HomePosRunFirstImp:=TRUE;
END_CASE
InternResetMode:=0;
(*###########################################################################*)
(* 	Einlesen der Tasten der Visualisierung	(CTS-Signal)										 *)
(*	--> Betriebsartenanwahl																									 *)
(*###########################################################################*)

IF 	BtnManual.PressedFlag THEN
	InternResetMode:=RESET_FOR_MANUAL;
END_IF

IF 	BtnStep.PressedFlag THEN
	CASE Mode OF
	MODE_STEP:
		;
	MODE_STEP_RUN,MODE_AUTO_STOP:
		Mode:=MODE_STEP_STOP;
	MODE_AUTO:
		Mode:=MODE_STEP;
	MODE_AUTO_RUN:
		Mode:=MODE_STEP_RUN;
	ELSE
		InternResetMode:=RESET_FOR_STEP;
	END_CASE
END_IF

IF 	BtnStepCycle.PressedFlag THEN
	CASE Mode OF
	MODE_STEP:
		Mode:=MODE_STEP_RUN;
	MODE_STEP_RUN,MODE_STEP_STOP,MODE_SPECIAL:
		InternNextStep:=TRUE;
	END_CASE
ELSE
	InternNextStep:=FALSE;
END_IF

IF 	BtnAuto.PressedFlag THEN
	CASE Mode OF
	MODE_STEP:
		Mode:=MODE_AUTO;
	MODE_STEP_RUN:
		Mode:=MODE_AUTO;
		StepToAuto:=TRUE;
	MODE_STEP_STOP:
		Mode:=MODE_AUTO_STOP;
		StepToAuto:=TRUE;
	MODE_AUTO,MODE_AUTO_RUN,MODE_AUTO_STOP:
		;
	ELSE
		InternResetMode:=RESET_FOR_AUTO;
	END_CASE
END_IF

IF 	BtnAutoStart.PressedFlag OR
	iRemoteAutoStart AND
	(BtnAuto.Visible OR BtnHomeRun.Visible)THEN
	IF 	BtnHomeRun.Visible OR
		Mode<=MODE_MANUAL AND NOT HomePosRunEnd THEN
		Mode:=MODE_HOME_POS_RUN;
  		HomePosRunFirstImp:=TRUE;
		InternLastMode:=MODE_AUTO_RUN;
		iRemoteAutoStart:=FALSE;
	ELSE
		Mode:=MODE_AUTO_RUN;
		StepToAuto:=FALSE;
		iRemoteAutoStart:=FALSE;
	END_IF
END_IF

IF 	BtnAutoStop.PressedFlag OR
 	iRemoteAutoStop AND BtnAutoStop.Visible THEN
	Mode:=MODE_AUTO_STOP;
	iRemoteAutoStop:=FALSE;
END_IF

IF 	BtnRunEmpty.PressedFlag OR gStartRunEmpty THEN
	gRunEmpty:=NOT(gRunEmpty);
END_IF

IF 	BtnHomeRun.PressedFlag THEN
	CASE Mode OF
	MODE_STEP:
		InternLastMode:=MODE_STEP;
		Mode:=MODE_HOME_POS_RUN;
		HomePosRunFirstImp:=TRUE;
	MODE_AUTO:

		InternLastMode:=MODE_AUTO;
		Mode:=MODE_HOME_POS_RUN;
		HomePosRunFirstImp:=TRUE;
	MODE_STEP_STOP:
		InternLastMode:=MODE_STEP;
		InternResetMode:=RESET_FOR_MODE_HOME_POS_RUN;
	MODE_AUTO_STOP:
		InternLastMode:=MODE_AUTO;
		InternResetMode:=RESET_FOR_MODE_HOME_POS_RUN;
	END_CASE
END_IF

IF 	BtnSpecial.PressedFlag THEN
	Mode:=MODE_SPECIAL;
	SpecialCycleEnd:=FALSE;
END_IF

IF 	BtnSpecStep.PressedFlag THEN
	TipInSpecialMode:=NOT(TipInSpecialMode);
END_IF
IF 	Mode<>MODE_SPECIAL THEN
	TipInSpecialMode:=FALSE;
END_IF

(*###########################################################################*)
(* Input-Variables - used from the application programmer										 *)
(* to modifie the mode out of a SFC 											 *)
(*###########################################################################*)
IF 	AskForNoMode THEN
	Mode:=MODE_NON;
	AskForNoMode:=FALSE;
	iRemoteAutoStart:=FALSE;
ELSIF
	AskForManual THEN
	InternResetMode:=RESET_FOR_MANUAL;
	AskForManual:=FALSE;
	iRemoteAutoStart:=FALSE;
ELSIF
	AskForStepMode THEN
	IF Mode<MODE_STEP THEN
		InternResetMode:=RESET_FOR_STEP;
	END_IF
	Mode:=MODE_STEP;
	AskForStepMode:=FALSE;
ELSIF
	AskForStepStart THEN
	IF 	Mode=MODE_STEP AND
		HomePosRunEnd THEN
		Mode:=MODE_STEP_RUN;
	END_IF
	AskForStepStart:=FALSE;
ELSIF
	AskForStepStop THEN
	Mode:=MODE_STEP_STOP;
	AskForStepStop:=FALSE;
ELSIF
	AskForAutoMode THEN
	IF Mode<MODE_STEP THEN
		InternResetMode:=RESET_FOR_AUTO;
	END_IF
	Mode:=MODE_AUTO;
	AskForAutoMode:=FALSE;
ELSIF
	AskForAutoStop THEN
	Mode:=MODE_AUTO_STOP;
	AskForAutoStop:=FALSE;
	iRemoteAutoStart:=FALSE;
ELSIF
	AskForAutoStart THEN
	IF 	Mode=MODE_AUTO AND
		HomePosRunEnd THEN
		Mode:=MODE_AUTO_RUN;
		StepToAuto:=FALSE;
	END_IF
	AskForAutoStart:=FALSE;
ELSIF
	AskForHomePos THEN
	AskForHomePos:=FALSE;
	CASE Mode OF
	MODE_STEP:
		InternLastMode:=MODE_STEP;
		Mode:=MODE_HOME_POS_RUN;
		HomePosRunFirstImp:=TRUE;
	MODE_AUTO:
		InternLastMode:=MODE_AUTO;
		Mode:=MODE_HOME_POS_RUN;
		HomePosRunFirstImp:=TRUE;
	MODE_STEP_STOP:
		InternLastMode:=MODE_STEP;
		InternResetMode:=RESET_FOR_MODE_HOME_POS_RUN;
	MODE_AUTO_STOP:
		InternLastMode:=MODE_AUTO;
		InternResetMode:=RESET_FOR_MODE_HOME_POS_RUN;
	END_CASE
ELSIF
	AskAutoStartOverHomePosRun THEN
	AskAutoStartOverHomePosRun:=FALSE;
	iRemoteAutoStart:=TRUE;
ELSIF
	AskForSpecialMode THEN
	InternResetMode:=RESET_FOR_AUTO;
	Mode:=MODE_SPECIAL;
	AskForSpecialMode:=FALSE;
END_IF

(*###########################################################################*)
(* Check the Key for SafetyDoor-ByPass
when it's put in -> MODE_AUTO_RUN change automaticaly to MODE_AUTO_STOP
when it's turnes -> mode change automaticaly to MODE_MANUAL 					 *)
(*###########################################################################*)
IF 	NOT ProtecKeyNotIn THEN
	CASE Mode OF
	MODE_AUTO_RUN:
		Mode:=MODE_AUTO_STOP;
	END_CASE
END_IF

IF NOT ProtecNotBridged THEN
	CASE Mode OF
	MODE_MANUAL,MODE_NON:
		;
	ELSE
		InternResetMode:=RESET_FOR_MANUAL;
	END_CASE
END_IF

IF	ControlOn AND
	MainValveOk AND
	SafetyDoorOk AND
	EmergencyOk AND
	BusControlState=STATE_OK AND
	UserOK THEN
	HardwareOk:=TRUE;
ELSE
	HardwareOk:=FALSE;
END_IF

IF 	InternResetMode>0 OR
	NOT HardwareOk THEN
	Mode:=MODE_NON;
END_IF

ControlIsOn:=HardwareOk;

(*###########################################################################*)
(* Für Visualisierung: Betriebsarten auf Bit legen													 *)
(*###########################################################################*)
CASE Mode OF
MODE_NON:
	sVisu.ManualOn:=FALSE;
	sVisu.StepOn:=FALSE;
	sVisu.AutoOn:=FALSE;
	sVisu.AutoStartOn:=FALSE;
	sVisu.AutoStopOn:=FALSE;
	sVisu.SpecialOn:=FALSE;
	sVisu.HomePosRunOn:=FALSE;
	sVisu.BasicManualMode:=FALSE;
	sVisu.BasicAutoMode:=FALSE;
	StepToAuto:=FALSE;

MODE_MANUAL:
	sVisu.ManualOn:=TRUE;
	sVisu.StepOn:=FALSE;
	sVisu.AutoOn:=FALSE;
	sVisu.AutoStartOn:=FALSE;
	sVisu.AutoStopOn:=FALSE;
	sVisu.HomePosRunOn:=FALSE;
	sVisu.SpecialOn:=FALSE;
	sVisu.BasicManualMode:=TRUE;
	sVisu.BasicAutoMode:=FALSE;
	StepToAuto:=FALSE;

MODE_STEP,MODE_STEP_RUN:
	sVisu.ManualOn:=FALSE;
	sVisu.StepOn:=TRUE;
	sVisu.AutoOn:=FALSE;
	sVisu.AutoStartOn:=FALSE;
	sVisu.AutoStopOn:=FALSE;
	sVisu.SpecialOn:=FALSE;
	sVisu.HomePosRunOn:=FALSE;
	sVisu.BasicManualMode:=FALSE;
	sVisu.BasicAutoMode:=TRUE;
	IF 	AskForAutoStop OR
		AskForStepStop THEN
		Mode:=MODE_STEP_STOP;
	END_IF

MODE_STEP_STOP:
	IF AutoCycleEnd THEN
		IF AskForAutoStop THEN
			InternResetMode:=RESET_FOR_MANUAL;
			Mode:=MODE_NON;
		ELSIF
			AskForStepStop THEN
			Mode:=MODE_STEP;
		ELSE
			Mode:=MODE_STEP;
		END_IF
	END_IF

MODE_AUTO:
	sVisu.ManualOn:=FALSE;
	sVisu.StepOn:=FALSE;
	sVisu.AutoOn:=TRUE;
	sVisu.AutoStartOn:=FALSE;
	sVisu.AutoStopOn:=FALSE;
	sVisu.HomePosRunOn:=FALSE;
	sVisu.SpecialOn:=TRUE;
	sVisu.BasicManualMode:=FALSE;
	sVisu.BasicAutoMode:=TRUE;

MODE_AUTO_RUN:
	sVisu.AutoStartOn:=TRUE;
	sVisu.AutoStopOn:=FALSE;
	IF AskForAutoStop THEN
		Mode:=MODE_AUTO_STOP;
	END_IF
	StepToAuto:=FALSE;

MODE_AUTO_STOP:
	sVisu.AutoStartOn:=FALSE;
	sVisu.AutoStopOn:=TRUE;
	IF AutoCycleEnd THEN
		IF NOT sInit.RemoteAutoStopToManual THEN
			Mode:=MODE_AUTO;
		ELSE
			Mode:=MODE_MANUAL;
		END_IF
	END_IF

MODE_HOME_POS_RUN:
	sVisu.ManualOn:=FALSE;
	sVisu.HomePosRunOn:=TRUE;
	sVisu.BasicManualMode:=FALSE;
	sVisu.BasicAutoMode:=TRUE;
	IF 	HomePosRunEnd THEN
		CASE InternLastMode OF
		MODE_STEP:
			Mode:=MODE_STEP;
		MODE_AUTO:
			Mode:=MODE_AUTO;
		MODE_AUTO_RUN: (*is used as next Mode*)
			Mode:=MODE_AUTO_RUN;
		ELSE
			Mode:=MODE_NON;
		END_CASE
	END_IF

MODE_SPECIAL:
	sVisu.SpecialOn:=TRUE;
	IF SpecialCycleEnd THEN
		Mode:=MODE_AUTO;
	END_IF
END_CASE
sVisu.RunEmptyOn:=gRunEmpty;

(*###########################################################################*)
(* Leerfahren zurücksetzen*)
(*###########################################################################*)
IF 	gRunEmpty AND
	RunEmptyEnd AND
	Mode=MODE_AUTO_RUN THEN
	gRunEmpty:=FALSE;
	RunEmptyEnd:=FALSE;
	Mode:=MODE_AUTO_STOP;
END_IF
IF 	gRunEmpty AND
	Mode<=MODE_MANUAL THEN
	gRunEmpty:=FALSE;
END_IF

(*###########################################################################*)
(* State des Betriebsartenbausteins zuweisen*)
(*###########################################################################*)
IF 	gInitOk AND
	gSetupOk THEN
	CASE Mode OF
		MODE_NON:
			IF	NOT ControlOn THEN
				State:=-2;						(* Steuerung einschalten!*)
			ELSE
				State:=-3;						(*Betriebsart anwählen!  *)
			END_IF
			(* SafetyDoor *)
			IF	NOT SafetyDoorOk THEN
				State:=-1;						(* Türe ist auf! *)
			END_IF
			(* MainValve *)
			IF NOT MainValveOk THEN
				State:=-7;						(* Hauptluft darf nicht ein sein!*)
			END_IF
			(* Emergency Stop*)
			IF NOT EmergencyOK THEN
				State:=-1;						(* Not-Aus betätigt! *)
			END_IF
			(* BusControl *)
			IF 	BusControlState<>STATE_OK THEN
				State:=-6;						(* Bus steht! *)
			END_IF
		MODE_MANUAL:
				State:=1;						(* Einzelbetrieb aktiv *)
		MODE_STEP:
			IF HomePosRunEnd THEN
				State:=2;							(* Tippbetrieb vorgewählt *)
			ELSE
				State:=-4;							(* Grundstellung fehlt *)
			END_IF
		MODE_STEP_RUN:
			State:=4;								(* Tippbetrieb läuft *)
		MODE_STEP_STOP:
			State:=10;								(* Tippbetrieb in letzten Zyklus *)
		MODE_AUTO:
			IF HomePosRunEnd THEN
				State:=3;							(* Automatikbetrieb vorgewählt *)
			ELSE
				State:=-4;							(* Grundstellung fehlt *)
			END_IF
		MODE_AUTO_RUN:
			State:=5;								(* Automatikbetrieb läuft *)
		MODE_AUTO_STOP:
			State:=6;								(* Automatikbetrieb im letzen Zyklus *)
		MODE_HOME_POS_RUN:
			State:=7;								(* Grundstellung wird angefahren *)
		MODE_SPECIAL:
			State:=8;								(* Spezialbetrieb läuft *)
	ELSE
			State:=0;								(* nicht definierter Status *)
	END_CASE
	IF 	NOT ProtecKeyNotIn THEN
		State:=16;									(* Schlüsselschalter ist gesteckt *)
	END_IF
	IF 	NOT ProtecNotBridged THEN
		State:=17;									(* Schutz ist überbrückt *)
	END_IF

ELSE
	State:=0;										(* nicht definierter Status *)
END_IF

(* copy input to output parameter *)
QProtecKeyNotIn		:= ProtecKeyNotIn;
QProtecNotBridged	:= ProtecNotBridged;
(*#################### Ende State zuweisen #################################*)
ErrorNo:=0;
ErrorText:='';
(*##########################################################################*)
(* Check home position																											*)
(* Pruefen der Grundstellung																								*)
(*##########################################################################*)
IF	NOT ProtecNotBridged THEN
	HomePositionInfoNo:=11;
ELSIF
	NOT ProtecKeyNotIn THEN
	HomePositionInfoNo:=10;
ELSE
	HomePositionInfoNo:=State_OK;
END_IF
(* Generating home position*)
(* Zuweisung der Grundstellung*)
IF 	HomePositionInfoNo=State_OK THEN
	HomePosition:=TRUE;
ELSE
	HomePosition:=FALSE;
END_IF
(* Objekt-Grundstellung verknüpfen mit GesamtGrundstellung *)
(* object-homeposition concat with mainhomeposition *)
gHomeOk:=gHomeOk AND HomePosition;

(*###########################################################################*)
(* Zuweisungen für Anzeigen am Display -> in sVisu. ...        															 *)
(*###########################################################################*)
(* buttons anzeigen *)
ShowButton:=HardwareOk;

BtnReset.Enable		:= TRUE;
BtnReset.Visible			:= Mode<=MODE_MANUAL;

BtnManual.Enable		:= ShowButton AND (DisableManualMode=FALSE OR Mode<=MODE_MANUAL) AND NOT(sInit.HideManualButton);
BtnManual.Visible		:= BtnManual.Enable;

BtnStep.Enable			:= ProtecNotBridged AND MainValveOk AND SafetyDoorOk AND NOT(Mode=MODE_SPECIAL) AND ShowButton;
BtnStep.Visible			:= BtnStep.Enable;

BtnStepCycle.Enable	:= (Mode=MODE_STEP OR Mode=MODE_STEP_RUN OR Mode=MODE_STEP_STOP OR TipInSpecialMode) AND NOT(BtnHomeRun.Visible) AND ShowButton AND NOT(sInit.HideNextStepButton);
BtnStepCycle.Visible		:= BtnStepCycle.Enable;

BtnAuto.Enable			:= ProtecNotBridged AND MainValveOk AND SafetyDoorOk AND NOT(Mode=MODE_SPECIAL) AND ShowButton;
BtnAuto.Visible			:= BtnAuto.Enable;

BtnAutoStart.Enable		:= (sVisu.AutoStartOn OR sVisu.AutoOn) AND
							Mode<>MODE_SPECIAL AND
							Mode<>MODE_AUTO_STOP AND
							(sInit.EnableQuickAutoStart OR NOT BtnHomeRun.Visible) AND
							ShowButton;
BtnAutoStart.Visible		:= BtnAutoStart.Enable;

BtnAutoStop.Enable		:= (Mode=MODE_AUTO_RUN OR Mode=MODE_AUTO_STOP) AND ShowButton;
BtnAutoStop.Visible		:= BtnAutoStop.Enable;

BtnRunEmpty.Enable	:= (Mode=MODE_AUTO_RUN OR Mode=MODE_AUTO_STOP OR Mode=MODE_AUTO) AND
						ShowBtnRunEmpty AND
						ShowButton AND
						NOT gRunEmpty;
BtnRunEmpty.Visible		:= Mode>MODE_MANUAL AND NOT BtnHomeRun.Visible;

BtnHomeRun.Enable	:= (	(Mode=MODE_AUTO OR Mode=MODE_STEP) AND
							NOT(HomePosRunEnd) OR
							Mode=MODE_HOME_POS_RUN OR
							Mode=MODE_AUTO_STOP OR
							Mode=MODE_STEP_STOP		) AND
							NOT(StepToAuto) AND
							ShowButton;
BtnHomeRun.Visible		:= BtnHomeRun.Enable;

BtnSpecial.Enable		:=  (Mode=MODE_AUTO AND NOT(BtnHomeRun.Visible) AND AutoCycleEnd AND HomePosRunEnd OR Mode=MODE_SPECIAL) AND ShowButton;
BtnSpecial.Visible		:= BtnSpecial.Enable;

BtnSpecStep.Enable		:= Mode=MODE_SPECIAL AND ShowButton;
BtnSpecStep.Visible		:=	BtnSpecStep.Enable;

(* interne Variablen *)
sVisu.State				:= State;
sVisu.HomePositionOk	:= HomePosRunEnd;
sVisu.HomePositionInfoNo:= HomePositionInfoNo;

(*###########################################################################*)
(* Zuweisen der Output-Variablen	        															 *)
(*###########################################################################*)
BasicManualMode	:= sVisu.BasicManualMode;
BasicAutoMode		:= sVisu.BasicAutoMode;
(*---------------------------------------------------------------------------
NextStep for StepMode and SemiAuotomaticMode 
Schrittweiterschaltung bei Tipp- und Teilautomatikbetrieb
  ---------------------------------------------------------------------------*)
CASE Mode OF
MODE_AUTO_RUN,MODE_AUTO_STOP,MODE_HOME_POS_RUN,MODE_SPECIAL:
	IF 	TipInSpecialMode THEN
		gTipImp:=InternNextStep;
	ELSE
		gTipImp:=TRUE;
	END_IF
ELSE
	gTipImp:=InternNextStep;
END_CASE
(*---------------------------------------------------------------------------
Reset for movements and functions 
Reset der Bewegungen und Funktionen
  ---------------------------------------------------------------------------*)

NoModeFirstImp(CLK:= (Mode=MODE_NON) );
ResetFlag(CLK:=NoModeFirstImp.Q OR BtnReset.Pressed);
QReset:=ResetFlag.Q;
ton_Reset(PT:= T#500ms, Q=>);

(*Reset für Tampondrucker*)
IF 	BtnReset.Pressed AND NOT ton_Reset.Q THEN
	ST00_72_K7.SetSignalHigh:=TRUE;
  	ton_Reset.IN := TRUE;
ELSIF
	ton_Reset.Q THEN
	ST00_72_K7.SetSignalLow:=TRUE;
	ton_Reset.IN := FALSE;
END_IF

(*---------------------------------------------------------------------------
Stop and Reset all sequences with : SFCInit-Flag 
Alle Schrittketten stoppen und zurücksetzen mit : SFCInit-Flag
  ---------------------------------------------------------------------------*)
CASE Mode OF
MODE_MANUAL,MODE_STEP_RUN,MODE_STEP_STOP,MODE_AUTO_RUN,MODE_AUTO_STOP,MODE_HOME_POS_RUN,MODE_SPECIAL:
	SFCInit:=FALSE;
MODE_AUTO:
	IF 	StepToAuto THEN
		SFCInit:=FALSE;
	ELSE
		SFCInit:=TRUE;
	END_IF
ELSE
	SFCInit:=TRUE;
END_CASE

(*---------------------------------------------------------------------------
Break to all sequences with : SFCPause-Flag 
Alle Schrittketten unterbrechen mit : SFCPause-Flag
  ---------------------------------------------------------------------------*)
IF 	NOT EnableFromPrevMach AND
	ProtecNotBridged THEN
	GlobalEnable:=FALSE;
	SFCTipMode:=TRUE;
	ErrorNo:=10;
	ErrorText:='Break from Previous Machine';
ELSIF
	NOT EnableFromNextMach AND
	ProtecNotBridged THEN
	GlobalEnable:=FALSE;
	SFCTipMode:=TRUE;
	ErrorNo:=11;
	ErrorText:='Break from Next Machine';
ELSE
	GlobalEnable:=TRUE;
	SFCTipMode:=FALSE;
END_IF

(*$$$$$$$$$$$$$$$$$$$$$$$$$$$$$$$$$$$$$$$$$$$$$$$$$$$$$$$$$$$$$$$$$$$$$$$$$$$
ErrorHandler
$$$$$$$$$$$$$$$$$$$$$$$$$$$$$$$$$$$$$$$$$$$$$$$$$$$$$$$$$$$$$$$$$$$$$$$$$$$*)
IF ErrorNo<>0 THEN
	;
END_IF

(*$$$$$$$$$$$$$$$$$$$$$$$$$$$$$$$$$$$$$$$$$$$$$$$$$$$$$$$$$$$$$$$$$$$$$$$$$$$
Reset of input variables.
$$$$$$$$$$$$$$$$$$$$$$$$$$$$$$$$$$$$$$$$$$$$$$$$$$$$$$$$$$$$$$$$$$$$$$$$$$$*)
DisableManualMode:=FALSE;
END_PROGRAM

(* POU Stations/ST_00/ST00_SFCs/_SpecialModeSFCs/SpecialMode03, SFC *)
PROGRAM SpecialMode03 (*Used for: Beschriften von Nest 1 - Einlegen nach Laser (Station 6) *)
VAR_OUTPUT
	SFCCurrentPOU		: STRING:='SpecialMode03';
	SFCCurrentStep	: STRING:='';
	SFCTime					:	DINT;
  State   				:	DINT;
  Result  				:	DINT;
END_VAR
VAR_INPUT
	Start						:	BOOL;
END_VAR
VAR
	MsgOK				:	BOOL;
	MsgCancel		:	BOOL;
	SFCRun					:	BOOL;
	SFCTimeStart		:	TIME;

	(* Userdefinded area *)

